	Components.P2_FixUnit
        .SuspendMoveWorkExpression( Components.P2_FixUnit.MoveWorkTask.Busy AND NOT inSafeCondition, '<#Movement is blocked due safe zone is interupted(robot in zone)#>');

    Components.P2_FixUnit
        .SuspendMoveHomeExpression(Components.P2_FixUnit.MoveHomeTask.Busy AND NOT inSafeCondition, '<#Movement is blocked due safe zone is interupted(robot in zone)#>');
END_IF;

IF _timerDisableSafety.Q THEN
	_temporarilyDisableSafety:=FALSE;
END_IF

PROPERTY Components : REFERENCE TO TcoPlbPaletizator_Components
GET
Components ref=_components;
END_GET
END_PROPERTY

(*~
	<docu>
		<summary>
			Gets the configuration of the MTS Pls feeder. 					
		</summary>			
	</docu>	
~*)
PROPERTY Config : REFERENCE TO TcoPlbPaletizator_Config_v_1_x_x
GET
Config REF= _config;
END_GET
END_PROPERTY

METHOD PUBLIC DefaultSignalisation
VAR_INPUT
END_VAR
Components.Q1_AttentionSignalisationR.Reset();
Components.Q2_AttentionSignalisationG.Reset();
Components.Q3_AttentionSignalisationB.Reset();

_blinker(inOffTime:=_config.BlinkTime,inOnTime:=_config.BlinkTime);
_timerEntryEmpty(in:= _status.EntryBufferEmpty,Pt:=_config.InfoTime);
_timerOutFull(in:=  _status.OutBufferFull ,Pt:=_config.InfoTime);
IF 
	NOT _timerEntryEmpty.Q
	AND NOT _timerOutFull.q THEN
	Components.Q2_AttentionSignalisationG.Set();
ELSIF  _blinker.IsOn THEN
	//all empty or disabled
//	IF NOT( NOT Components.I2_iBuffer1IsReadyToLoad.Signal
//		XOR NOT _config.Buffer1Disabled)
//		AND 
//		NOT(NOT Components.I4_iBuffer2IsReadyToLoad.Signal
//		XOR NOT _config.Buffer2Disabled)
//		AND
//		NOT( NOT Components.I6_iBuffer3IsReadyToLoad.Signal
//		XOR NOT _config.Buffer3Disabled)
//		AND 
//		NOT( NOT Components.I8_iBuffer4IsReadyToLoad.Signal
//		XOR NOT _config.Buffer4Disabled)
		
//		 THEN
//		Components.Q1_AttentionSignalisationR.Set();
	IF inLightCurtainOk AND 
		(
		THIS^._feedNewBlisterTask.Busy
		OR
		THIS^._throwBlisterTask.Busy
		)THEN
		Messenger.Warning('<#CAKANIE NA OBSLUHU PALETIZERA - NARUSENA SVETELNA BRANA!#>');
		Components.Q1_AttentionSignalisationR.Set();
		Components.Q2_AttentionSignalisationG.Set();
	ELSIF _timerEntryEmpty.Q
		THEN
		Components.Q1_AttentionSignalisationR.Set();
		Components.Q2_AttentionSignalisationG.Set();
	ELSIF _timerOutFull.Q
		THEN
		
		Components.Q1_AttentionSignalisationR.Set();
		Components.Q2_AttentionSignalisationG.Set();
	
//	ELSIF NOT _status.OutBufferFull
//		AND _status.EntryBufferEmpty 
//		AND NOT _status.BlisterReady THEN	
//		Components.Q1_AttentionSignalisationR.Set();
//	ELSIF  _status.OutBufferFull  THEN
//		Components.Q1_AttentionSignalisationR.Set();	
	
	END_IF;


	
END_IF;
END_METHOD

METHOD PUBLIC FeedNewBlister : TcoCore.ITcoTaskStatus

FeedNewBlister := _feedNewBlisterTask.Invoke();
END_METHOD

PROPERTY FeedNewBlisterTask : REFERENCE TO TcoFeedingSequenceTask
GET
FeedNewBlisterTask ref=_feedNewBlisterTask;
END_GET
END_PROPERTY

METHOD PUBLIC LoaadPositions : BOOL
VAR_INPUT
END_VAR
LoaadPositions:= Components.Manipulator.LoadPositionsTask.WithId(_config.PositionsSetName).Invoke().Done and Components.Manipulator.LoadPositionsTask.ReadSuccessfuly ;
END_METHOD

PROPERTY OutBufferFull : bool
GET
OutBufferFull:=_status.OutBufferFull;
END_GET
END_PROPERTY

PROPERTY ReadyToUnloadComponent : bool
GET
ReadyToUnloadComponent:=_status.ReadyToUnloadComponents;
END_GET
END_PROPERTY

(*~
	<docu>
		<summary>
			Restores this instance to the Ready state. Can be called explicitly or from within one of the restore mechanisms.	
		</summary>			
	</docu>	
~*)
METHOD  Restore : ITcoRestorable
_components.Manipulator.Restore();
_feedNewBlisterTask.Restore();
_throwBlisterTask.Restore();
_setToDefaultTask.Restore();
_messenger.UnPin();
END_METHOD

METHOD PRIVATE SequenceIncomingBlister
VAR_INPUT
	refSequenceTask : REFERENCE TO TcoFeedingSequenceTask;
	
	
END_VAR

VAR
    seq    : REFERENCE TO TcoCore.TcoSequence;


END_VAR

VAR_INST
	_timer:ton;
	_moveParam: TcoSingleAxisMoveParam;

END_VAR
seq REF= refSequenceTask.Sequence;
refSequenceTask(inoStatus := _status, inoConfig := _config);

IF NOT Components.I1_iBuffer1HasNotCriticalLevel.Signal AND NOT _config.Buffer1Disabled THEN
    Messenger.Warning('<#Buffer 1  minimalne mnozstvo!#>');
END_IF

IF NOT Components.I3_iBuffer2HasNotCriticalLevel.Signal AND NOT _config.Buffer2Disabled THEN
    Messenger.Warning('<#Buffer 2 minimalne mnozstvo!#>');
END_IF

IF NOT Components.I5_iBuffer3HasNotCriticalLevel.Signal AND NOT _config.Buffer3Disabled THEN
    Messenger.Warning('<#Buffer 3 minimalne mnozstvo!#>');
END_IF

IF NOT Components.I7_iBuffer4HasNotCriticalLevel.Signal AND NOT _config.Buffer4Disabled THEN
    Messenger.Warning('<#Buffer 4 minimalne mnozstvo!#>');
END_IF

seq.Open();
seq.Observer := refSequenceTask.Observer;

//***************************************************************************************************     
//    This step will be executed and immediately finished, as the condition in Await method is true.
IF seq.Step(0, TRUE, '<#INIT#>') THEN
    Messenger.Warning('<#BEZPECNOST ZARIADENIA NARUSENA. NIEJE MOZNE VYKONAT AKCIU#>');
    IF _status.SafeCondition THEN
        seq.CompleteStep();
    END_IF;
END_IF

//***************************************************************************************************     

//***************************************************************************************************     
IF seq.Step(20, TRUE, '<#ZASUNUTIE POZICNEJ JEDNOTKY#>') THEN

    seq.StepCompleteWhen( (*Components.P2_FixUnit.MoveToWork().Done OR*)
        Components.I11_BlisterInWorkPosition.IsFalse AND_THEN Components.P1_PositionUnit.MoveToHome().Done);

END_IF

//***************************************************************************************************     

//IF (seq.Step(inStepID := 25,
//    inEnabled := TRUE,
//    inStepDescription := 'LOAD CREATED POSITIONS')) THEN
//    //--------------------------------------------------------   
//    IF Seq.IsFreshState THEN
//        Components.Manipulator.Restore();
//    END_IF

//    IF Components.Manipulator.LoadPositionsTask.WithId(_config.PositionsSetName).Invoke().Done AND
//        Components.Manipulator.LoadPositionsTask.ReadSuccessfuly THEN
//        seq.CompleteStep();
//    END_IF

//    //--------------------------------------------------------			
//END_IF

//***************************************************************************************************     
IF seq.Step(30, TRUE, '<#KONTROLA STAVU ZASOBNIKOV') THEN

    IF Components.I2_iBuffer1IsReadyToLoad.IsTrue AND NOT _config.Buffer1Disabled THEN
        _requiredPosition := _positions.LoadFromBuffer1Pos;
        seq.StepCompleteWhen(TRUE);

    ELSIF Components.I4_iBuffer2IsReadyToLoad.Istrue AND NOT _config.Buffer2Disabled THEN
        _requiredPosition := _positions.LoadFromBuffer2Pos;
        seq.StepCompleteWhen(TRUE);

    ELSIF Components.I6_iBuffer3IsReadyToLoad.IsTrue AND NOT _config.Buffer3Disabled THEN
        _requiredPosition := _positions.LoadFromBuffer3Pos;
        seq.StepCompleteWhen(TRUE);

    ELSIF Components.I8_iBuffer4IsReadyToLoad.IsTrue AND NOT _config.Buffer4Disabled THEN
        _requiredPosition := _positions.LoadFromBuffer4Pos;
        seq.StepCompleteWhen(TRUE);
    ELSE
        IF _config.Buffer1Disabled AND _config.Buffer2Disabled AND _config.Buffer3Disabled AND _config.Buffer4Disabled THEN
            Messenger.Error('<#VSETKY ZASDOBNIKY SU VYPNUTE !!!#>');
        ELSE
            Messenger.Error('<#CHYBA ZASOBNIKY SU PRAZDNE !!!#>');

        END_IF
    END_IF
END_IF

//***************************************************************************************************     

//***************************************************************************************************     
IF seq.Step(34, TRUE, 'RESET MANIPULATORA') THEN
    IF Seq.IsFreshState OR NOT inLightCurtainOk THEN
        Components.Manipulator.Restore();
    END_IF

    IF inLightCurtainOk THEN

        IF Components.Manipulator.ResetDrive().Done AND_THEN
            Components.Manipulator.SoeReset().Done AND_THEN
            NOT Components.Manipulator.Axis.AxisStatus.Error THEN
            seq.CompleteStep();
        END_IF;
    END_IF
END_IF

//***************************************************************************************************     

//***************************************************************************************************     
IF seq.Step(35, TRUE, 'RESET MANIPULATORA') THEN
    //    IF seq.CurrentStep.Duration >= T#2S THEN
    //        seq.RequestStep(34);

    //    END_IF

    //    seq.StepCompleteWhen(Components.Manipulator.Initialize());
    Seq.CompleteStep();
END_IF

//***************************************************************************************************     

//***************************************************************************************************     
IF seq.Step(40, TRUE, 'PRESUN MANIPULATORA - NOVY BLISTER') THEN
    IF Seq.IsFreshState THEN
        Components.Manipulator.Restore();
    END_IF

    IF Components.Manipulator.Axis.AxisStatus.Error OR Components.Manipulator.Axis.AxisStatus.Disabled THEN
        seq.RequestStep(34);
    END_IF

    _moveParam.Position := _requiredPosition.Axis1.Position;
    _moveParam.Velocity := _requiredPosition.Axis1.Velocity;
    _moveParam.Acceleration := _requiredPosition.Axis1.Acceleration;
    _moveParam.Deceleration := _requiredPosition.Axis1.Deceleration;
    _moveParam.Jerk := _requiredPosition.Axis1.Jerk;

    IF Components.Manipulator.MoveAbsolute(_moveParam).Done THEN
        seq.CompleteStep();
    END_IF

END_IF

//***************************************************************************************************     

//***************************************************************************************************     
IF seq.Step(45, TRUE, 'KONTROLA BLISTRA VO FIXTURE') THEN

    Messenger.OnCondition(NOT Components.I12_BlisterPickedCorrectly.Signal).Error('<#KOLIZNY STAV SKONTROLUJTE BLISTRE!!!#>');

    seq.StepCompleteWhen(COmponents.I11_BlisterInWorkPosition.IsFalse);

END_IF

//***************************************************************************************************     

//***************************************************************************************************     
IF seq.Step(50, TRUE, 'VYSUNUTIE POZICNEJ JEDNOTKY') THEN
    IF seq.IsFreshState THEN
        _timer(IN := FALSE);
    END_IF

    _timer(IN := Components.P1_PositionUnit.MoveToWork().Done, PT := _config.StabilisationTime);
    seq.StepCompleteWhen(Components.P2_FixUnit.MoveToHome().Done AND_THEN Components.P1_PositionUnit.MoveToWork().Done AND _timer.Q);

END_IF

//***************************************************************************************************     

//***************************************************************************************************     
IF seq.Step(60, TRUE, 'UPEVNENIE BLISTRA') THEN
    IF seq.IsFreshState THEN
        _timer(IN := FALSE);
    END_IF

    _timer(IN := Components.P2_FixUnit.MoveToWork().Done, PT := _config.StabilisationTime);

    seq.StepCompleteWhen(_timer.Q);
END_IF

//***************************************************************************************************     

//***************************************************************************************************     
IF seq.Step(70, TRUE, 'ZASUNUTIE POZICNEJ JEDNOTKY A KONTROLA BLISTRA') THEN
    Messenger.OnCondition(Components.P1_PositionUnit.AtHome AND NOT Components.I11_BlisterInWorkPosition.Signal)
        .Error('NEPODARILO SA ODOBRAT BLISTER (PLNY)!');

    Messenger.OnCondition(Components.P1_PositionUnit.AtHome AND
            NOT Components.I12_BlisterPickedCorrectly.Signal).Error('<#KOLIZNY STAV SKONTROLUJTE BLISTRE!!!#>');

    IF Components.P1_PositionUnit.MoveToHome().Done AND_THEN
        Components.I11_BlisterInWorkPosition.IsTrue AND
        Components.I12_BlisterPickedCorrectly.IsTrue THEN
        seq.RequestStep(75);
    END_IF
END_IF

//***************************************************************************************************     
//***************************************************************************************************     
IF seq.Step(74, TRUE, 'RESET MANIPULATORA') THEN
    IF Seq.IsFreshState or not inLightCurtainOk THEN
        Components.Manipulator.Restore();
    END_IF

    IF inLightCurtainOk THEN
        IF Components.Manipulator.ResetDrive().Done AND_THEN
            Components.Manipulator.SoeReset().Done AND_THEN
            NOT Components.Manipulator.Axis.AxisStatus.Error THEN
            seq.CompleteStep();
        END_IF;
    END_IF;
END_IF

//***************************************************************************************************     

//***************************************************************************************************     
IF seq.Step(75, TRUE, 'RESET MANIPULATORA') THEN
    //    IF seq.CurrentStep.Duration >= T#2S THEN
    //        seq.RequestStep(34);

    //    END_IF

    //    seq.StepCompleteWhen(Components.Manipulator.Initialize());
    Seq.CompleteStep();
END_IF

//***************************************************************************************************     

//***************************************************************************************************     
IF seq.Step(80, TRUE, ' PRESUN MANIPULATORA - VYLOZENIE PRAZDNY BLISTER') THEN
    IF Seq.IsFreshState THEN
        Components.Manipulator.Restore();
    END_IF

    IF Components.Manipulator.Axis.AxisStatus.Error OR Components.Manipulator.Axis.AxisStatus.Disabled THEN
        seq.RequestStep(74);
    END_IF

    _requiredPosition := _positions.WorkPos;
    _moveParam.Position := _requiredPosition.Axis1.Position;
    _moveParam.Velocity := _requiredPosition.Axis1.Velocity;
    _moveParam.Acceleration := _requiredPosition.Axis1.Acceleration;
    _moveParam.Deceleration := _requiredPosition.Axis1.Deceleration;
    _moveParam.Jerk := _requiredPosition.Axis1.Jerk;

    IF Components.Manipulator.MoveAbsolute(_moveParam).Done THEN
        seq.CompleteStep();
    END_IF

END_IF

//***************************************************************************************************     
IF seq.Step(90, TRUE, 'VYSUNUTIE POZICNEJ JEDNOTKY') THEN

    seq.StepCompleteWhen(Components.P1_PositionUnit.MoveToWork().Done);

END_IF

//***************************************************************************************************     

IF (seq.Step(inStepID := seq.RESTORE_STEP_ID,
    inEnabled := TRUE,
    inStepDescription := 'RETURN TO THE START OF THE SEQUENCE')) THEN
    //--------------------------------------------------------	
    refSequenceTask.DoneWhen(TRUE);
    seq.CompleteSequence();
    //--------------------------------------------------------			
END_IF;

IF refSequenceTask.HandleTaskError() THEN
    //here we can decide what to do
    //	refSequenceTask.Restore();
    _feedNewBlisterTask.Restore();
END_IF

seq.Close();
END_METHOD

METHOD PRIVATE SequenceOutgoingBlister
VAR_INPUT
	refSequenceTask : REFERENCE TO TcoFeedingSequenceTask;
	
	
END_VAR

VAR
    seq    : REFERENCE TO TcoCore.TcoSequence;

END_VAR

VAR_INST
	_timer:ton;
	_timerOptional:ton;
	_moveParam: TcoSingleAxisMoveParam;

END_VAR
seq REF= refSequenceTask.Sequence;
refSequenceTask(inoStatus := _status, inoConfig := _config);

IF Components.I9_iThrowBuffer1Isfull.Signal AND NOT _config.EmptyBuffer1Disabled THEN
    Messenger.Warning('<#VYSTUPNY ZASOBNIK 1 PLNY(BUFFER) !!!#>');
END_IF

IF Components.I10_iThrowBuffer2Isfull.Signal AND NOT _config.EmptyBuffer2Disabled THEN
    Messenger.Warning('<#VYSTUPNY ZASOBNIK 2 PLNY(BUFFER) !!!#>');
END_IF

seq.Open();
seq.Observer := refSequenceTask.Observer;

//***************************************************************************************************     
//    This step will be executed and immediately finished, as the condition in Await method is true.
IF seq.Step(0, TRUE, '<#INIT#>') THEN
    Messenger.Warning('<#BEZPECNOST ZARIADENIA NARUSENA. NIEJE MOZNE VYKONAT AKCIU#>');
    IF _status.SafeCondition THEN
        seq.CompleteStep();
    END_IF;
END_IF

//***************************************************************************************************     

//***************************************************************************************************     
IF seq.Step(10, TRUE, 'ZASUNUTIE POZICNEJ JEDNOTKY') THEN

    seq.StepCompleteWhen((Components.P2_FixUnit.MoveToWork().Done OR Components.I11_BlisterInWorkPosition.IsFalse) AND_THEN
            Components.P1_PositionUnit.MoveToHome().Done);

END_IF

//***************************************************************************************************     

//IF (seq.Step(inStepID := 25,
//    inEnabled := TRUE,
//    inStepDescription := 'LOAD CREATED POSITIONS')) THEN
//    //--------------------------------------------------------   
//    IF Seq.IsFreshState THEN
//        Components.Manipulator.Restore();
//    END_IF

//    IF Components.Manipulator.LoadPositionsTask.WithId(_config.PositionsSetName).Invoke().Done AND
//        Components.Manipulator.LoadPositionsTask.ReadSuccessfuly THEN
//        seq.CompleteStep();
//    END_IF

//    //--------------------------------------------------------			
//END_IF

//***************************************************************************************************     

//***************************************************************************************************     
IF seq.Step(20, TRUE, 'KONTROLA ZASOBNIKOU PRE PRAZDNE BLISTRE') THEN

    Messenger.OnCondition(Components.I9_iThrowBuffer1Isfull.Signal AND NOT _config.EmptyBuffer1Disabled)
        .Warning('<#Zasobnik 1 na prazdne blistre plny!#>');

    Messenger.OnCondition(Components.I10_iThrowBuffer2Isfull.Signal AND NOT _config.EmptyBuffer2Disabled)
        .Warning('<#Zasobnik 2 na prazdne blistre plny!#>');

    IF Components.I9_iThrowBuffer1Isfull.IsFalse AND NOT _config.EmptyBuffer1Disabled THEN
        _requiredPosition := _positions.UnloadEmpty1Postion;
        seq.StepCompleteWhen(TRUE);

    ELSIF Components.I10_iThrowBuffer2Isfull.IsFalse AND NOT _config.EmptyBuffer2Disabled THEN
        _requiredPosition := _positions.UnloadEmpty2Postion;
        seq.StepCompleteWhen(TRUE);
    ELSE
        IF _config.EmptyBuffer1Disabled AND _config.EmptyBuffer2Disabled THEN
            Messenger.Error('<#ZASDOBNIKY PRE PRAZDNE BLISTRE SU VYPNUTE !!!#>');
        ELSE
            Messenger.Error('<#CHYBA ZASOBNIKY NA PRAZDNE BLISTRE OBSADENE !!!#>');

        END_IF
    END_IF;

END_IF

//***************************************************************************************************     

//***************************************************************************************************     
IF seq.Step(34, TRUE, 'RESET MANIPULATORA') THEN
    IF Seq.IsFreshState or not inLightCurtainOk THEN
        Components.Manipulator.Restore();
    END_IF

    IF inLightCurtainOk THEN
        IF Components.Manipulator.ResetDrive().Done AND_THEN
            Components.Manipulator.SoeReset().Done AND_THEN
            NOT Components.Manipulator.Axis.AxisStatus.Error THEN
            seq.CompleteStep();
        END_IF;
    END_IF;
END_IF

//***************************************************************************************************     

//***************************************************************************************************     
IF seq.Step(35, TRUE, 'RESET MANIPULATORA') THEN
    //    IF seq.CurrentStep.Duration >= T#2S THEN
    //        seq.RequestStep(34);

    //    END_IF

    //    seq.StepCompleteWhen(Components.Manipulator.Initialize());
    Seq.CompleteStep();
END_IF

//***************************************************************************************************     

//***************************************************************************************************     
IF seq.Step(40, TRUE, 'PRESUN MANIPULATORA - NOVY BLISTER') THEN
    IF Seq.IsFreshState THEN
        Components.Manipulator.Restore();
    END_IF

    IF Components.Manipulator.Axis.AxisStatus.Error OR Components.Manipulator.Axis.AxisStatus.Disabled THEN
        seq.RequestStep(34);
    END_IF

    _moveParam.Position := _requiredPosition.Axis1.Position;
    _moveParam.Velocity := _requiredPosition.Axis1.Velocity;
    _moveParam.Acceleration := _requiredPosition.Axis1.Acceleration;
    _moveParam.Deceleration := _requiredPosition.Axis1.Deceleration;
    _moveParam.Jerk := _requiredPosition.Axis1.Jerk;

    IF Components.Manipulator.MoveAbsolute(_moveParam).Done THEN
        seq.CompleteStep();
    END_IF

END_IF

//***************************************************************************************************    

//***************************************************************************************************     
IF seq.Step(43, TRUE, 'VYLOZENIE PRAZDNEHO BLISTRA DO ZASOBNIKA PRESUN POZICNEJ JEDNOTKY') THEN
    IF seq.IsFreshState THEN
        _timer(IN := FALSE);
    END_IF

    _timer(IN := Components.P1_PositionUnit.MoveToWork().Done, PT := _config.StabilisationTime);

    seq.StepCompleteWhen(_timer.Q);

END_IF

//***************************************************************************************************     
IF seq.Step(45, TRUE, 'VYLOZENIE PRAZDNEHO BLISTRA DO ZASOBNIKA') THEN
    IF seq.IsFreshState THEN
        _timer(IN := FALSE);
        _timerOptional(IN := FALSE);
    END_IF

    _timer(IN := Components.P2_FixUnit.MoveToHome().Done, PT := _config.StabilisationTime);
    _timerOptional(IN := Components.I11_BlisterInWorkPosition.IsFalse, PT := _config.StabilisationTime);

    seq.StepCompleteWhen(_timer.Q OR _timerOptional.Q);
END_IF

//***************************************************************************************************     
IF seq.Step(50, TRUE, 'VYLOZENIE PRAZDNEHO BLISTRA DO ZASOBNIKA') THEN

    seq.StepCompleteWhen(Components.P1_PositionUnit.MoveToHome().Done);

END_IF

//*************************************************************************************************** 

//***************************************************************************************************     
IF seq.Step(60, TRUE, 'KONTROLA VYLOZENIA BLISTRA DO  ZASOBNIKA (PRAZDNE)') THEN
    Messenger.Error('NEPODARILO SA VYLOZIT PRAZDNY BLISTER!');
    seq.StepCompleteWhen(Components.I11_BlisterInWorkPosition.IsFalse);

END_IF

//*************************************************************************************************** 

IF (seq.Step(inStepID := seq.RESTORE_STEP_ID,
    inEnabled := TRUE,
    inStepDescription := 'RETURN TO THE START OF THE SEQUENCE')) THEN
    //--------------------------------------------------------	
    refSequenceTask.DoneWhen(TRUE);
    seq.CompleteSequence();
    //--------------------------------------------------------			
END_IF;

IF refSequenceTask.HandleTaskError() THEN
    //here we can decide what to do
    //	refSequenceTask.Restore();
    _throwBlisterTask.Restore();

END_IF

seq.Close();
END_METHOD

METHOD PRIVATE SequenceSetToDefault
VAR_INPUT
	refSequenceTask : REFERENCE TO TcoFeedingSequenceTask;
	inResetOnlyManipulator:BOOL;
	
END_VAR

VAR
    seq    : REFERENCE TO TcoCore.TcoSequence;

END_VAR

VAR_INST
	_timer:ton;
	
END_VAR
seq REF= refSequenceTask.Sequence;
refSequenceTask(inoStatus:=_status,inoConfig:=_config);
seq.Open();
seq.Observer := refSequenceTask.Observer;



		



//***************************************************************************************************     
//    This step will be executed and immediately finished, as the condition in Await method is true.
IF seq.Step(0,TRUE,'<#INIT#>') THEN   
	Messenger.Warning('<#BEZPECNOST ZARIADENIA NARUSENA. NIEJE MOZNE VYKONAT AKCIU#>');     
	IF _status.SafeCondition THEN
    	seq.CompleteStep();
	END_IF;
END_IF        
//***************************************************************************************************     



//***************************************************************************************************     
IF seq.Step(10,NOT inResetOnlyManipulator,'<#VYCHODIZA POLOHA - ZASUNUTIE POZICIEJ JEDNOTKY P1 #>') THEN   

    seq.StepCompleteWhen(Components.P1_PositionUnit.MoveToHome().Done );
END_IF        
//***************************************************************************************************   


//***************************************************************************************************     
IF seq.Step(20,not inResetOnlyManipulator,'<#VYCHODIZA POLOHA - ZASUNUTIE UPEVNENIA BLISTRA  P2#>') THEN   

    seq.StepCompleteWhen(Components.P2_FixUnit.MoveToHome().Done);
END_IF        
//***************************************************************************************************   


//***************************************************************************************************     
IF (seq.Step(inStepID := 30,
    inEnabled := TRUE,
    inStepDescription := 'LOAD POSITIONS FROM DB')) THEN
    //--------------------------------------------------------   
    IF Seq.IsFreshState THEN
        Components.Manipulator.Restore();
    END_IF

    IF Components.Manipulator.LoadPositionsTask.WithId(_config.PositionsSetName).Invoke().Done AND
        Components.Manipulator.LoadPositionsTask.ReadSuccessfuly THEN
        seq.CompleteStep();
    END_IF

    //--------------------------------------------------------			
END_IF      

//***************************************************************************************************     
IF seq.Step(40, TRUE, 'RESET MANIPULATORA') THEN
    IF Seq.IsFreshState THEN
        Components.Manipulator.Restore();
    END_IF

    IF Components.Manipulator.ResetDrive().Done AND_THEN
        Components.Manipulator.SoeReset().Done AND_THEN
        NOT Components.Manipulator.Axis.AxisStatus.Error THEN
        seq.CompleteStep();
    END_IF;
END_IF

//***************************************************************************************************     




IF (seq.Step(inStepID := seq.RESTORE_STEP_ID,
    inEnabled := TRUE,
    inStepDescription := 'RETURN TO THE START OF THE SEQUENCE')) THEN
    //--------------------------------------------------------	
		refSequenceTask.DoneWhen(TRUE);
    	seq.CompleteSequence();
    //--------------------------------------------------------			
END_IF;



IF refSequenceTask.HandleTaskError() THEN
	
	//here we can decide what to do
	//	refSequenceTask.Restore();

END_IF

seq.Close();
END_METHOD

(*~
	<docu>
		<summary>
		    Custom service (manual, maintenance) logic.
			This method must be implemented in derived class.
		</summary>			
	</docu>	
~*)
METHOD PROTECTED  ServiceMode
_components.Q3_AttentionSignalisationB.Service();
_components.Q2_AttentionSignalisationG.Service();
_components.Q1_AttentionSignalisationR.Service();
_components.P2_FixUnit.Service();
_components.P1_PositionUnit .Service();
_components.Manipulator.Service();
END_METHOD

PROPERTY PUBLIC SetSequencesToStep : bool
GET
SetSequencesToStep:=_setSequencesToStep;
END_GET
SET
_setSequencesToStep:=SetSequencesToStep;
END_SET
END_PROPERTY

METHOD PUBLIC SetToDefault : TcoCore.ITcoTaskStatus

VAR
	inResetOnlyManipulator:BOOL;
END_VAR
_control.ResetOnlyManipulator:=inResetOnlyManipulator;
SetToDefault := _setToDefaultTask.Invoke();
END_METHOD

PROPERTY SetToDefaultTask : REFERENCE TO TcoFeedingSequenceTask
GET
SetToDefaultTask ref=_setToDefaultTask;
END_GET
END_PROPERTY

(*~
	<docu>
		<summary>
			Gets the status of the MTS Pls feeder. 					
		</summary>			
	</docu>	
~*)
PROPERTY Status : REFERENCE TO TcoPlbPaletizator_Status_v_1_x_x
GET
Status REF= _status;
END_GET
END_PROPERTY

METHOD PUBLIC ThrowBlister : TcoCore.ITcoTaskStatus

ThrowBlister := _throwBlisterTask.Invoke();
END_METHOD

PROPERTY ThrowBlisterTask : REFERENCE TO TcoFeedingSequenceTask
GET
ThrowBlisterTask ref=_throwBlisterTask;
END_GET
END_PROPERTY

END_FUNCTION_BLOCK

// ---- Abstractions/Components/MtsFeeding/TcoFeedingSequenceTask.TcPOU
FUNCTION_BLOCK  TcoFeedingSequenceTask EXTENDS TcoCore.TcoTask
VAR_IN_OUT
	inoStatus:TcoFeeding_Status_v_1_x_x;
	inoConfig:TcoFeeding_Config_v_1_x_x;

END_VAR
VAR
	_sequence      : TcoCore.TcoSequence(THIS^, eRestoreMode.None);
    _observerSequence       : TcoCore.TcoSequencerObserver(THIS^);
	_infoTime:TIME;
	_errorTime:	TIME;
	_errorMessage:TcoCore.TcoMessenger(THIS^);

END_VAR

IF  __ISVALIDREF(inoConfig) THEN  
_infoTime := THIS^.inoConfig.InfoTime;
_errorTime := THIS^.inoConfig.ErrorTime;
END_IF;

PROPERTY PUBLIC ErrorTime : REFERENCE TO TIME
GET
ErrorTime REF=_errorTime;
END_GET
END_PROPERTY

METHOD PUBLIC HandleTaskError :BOOL;
VAR_INPUT
END_VAR
IF THIS^.ElapsedTime > THIS^.ErrorTime AND THIS^.ErrorTime<>T#0S THEN
	THIS^.ThrowWhen(TRUE);
END_IF

HandleTaskError := THIS^.Error AND NOT THIS^._errorMessage.Pinned;
END_METHOD

PROPERTY InfoTime :REFERENCE TO TIME
GET
InfoTime REF=_infoTime;
END_GET
END_PROPERTY

PROPERTY PUBLIC Observer : REFERENCE TO TcoCore.TcoSequencerObserver
GET
Observer ref=_observerSequence;
END_GET
END_PROPERTY

METHOD PROTECTED OnError
VAR
	description: STRING;
END_VAR
description := '<#Task finished with error.#>'; 
IF  __ISVALIDREF(inoStatus) THEN   THIS^.inoStatus.ActionDescription := description; END_IF;
THIS^._errorMessage.Error('To restore acknowledge this alarm.').Pin();
END_METHOD

(*~
	<docu>
		<summary>
			Restores this instance to the Ready state. Can be called explicitly or from within one of the restore mechanisms.
			<para>
				See also <see cref="PlcDocu.TcoCore.TcoTask.AutoRestorable()"/>
			</para>
		</summary>			
	</docu>	
~*)
METHOD Restore : ITcoRestorable
SUPER^.Restore();
_sequence.ModeController.Mode :=eSequencerMode.CyclicMode;
_messenger.UnPin();
_errorMessage.UnPin();
_sequence.Restore();
END_METHOD

PROPERTY PUBLIC Sequence : REFERENCE TO TcoCore.TcoSequence
GET
Sequence ref=_sequence;
END_GET
END_PROPERTY

METHOD SetCyclicMode
VAR_INPUT
END_VAR
_sequence.ModeController.Mode :=eSequencerMode.CyclicMode;
END_METHOD

METHOD SetStepMode
VAR_INPUT
END_VAR
_sequence.ModeController.Mode :=eSequencerMode.StepMode;
END_METHOD

END_FUNCTION_BLOCK

// ---- Abstractions/Components/MtsFeeding/Blisters/Plb/TcoPlbPaletizator_Positions.TcPOU
FUNCTION_BLOCK TcoPlbPaletizator_Positions EXTENDS TcoDrivesBeckhoff.TcoSingleAxisPositionsRootContainer
VAR_INPUT
END_VAR
VAR_OUTPUT
END_VAR
VAR

	
	{attribute addProperty Name "<#Pracovna pozicia#>"}
	WorkPosition : TcoDrivesBeckhoff.TcoMultiAxisMoveParam;
	{attribute addProperty Name "<#Naberacia pozicia Buffer1#>"}
	LoadFromBuffer1Postion : TcoDrivesBeckhoff.TcoMultiAxisMoveParam;
	{attribute addProperty Name "<#Naberacia pozicia Buffer2#>"}
	LoadFromBuffer2Postion : TcoDrivesBeckhoff.TcoMultiAxisMoveParam;
	{attribute addProperty Name "<#Naberacia pozicia Buffer3#>"}
	LoadFromBuffer3Postion : TcoDrivesBeckhoff.TcoMultiAxisMoveParam;
	{attribute addProperty Name "<#Naberacia pozicia Buffer4#>"}
	LoadFromBuffer4Postion : TcoDrivesBeckhoff.TcoMultiAxisMoveParam;
	{attribute addProperty Name "<#Vykladacia pozicia pre prazdne blistre 1#>"}
	UnloadEmpty1Postion : TcoDrivesBeckhoff.TcoMultiAxisMoveParam;
	{attribute addProperty Name "<#Vykladacia pozicia pre prazdne blistre 2#>"}
	UnloadEmpty2Postion : TcoDrivesBeckhoff.TcoMultiAxisMoveParam;

END_VAR

PROPERTY PUBLIC LoadFromBuffer1Pos : reference to TcoDrivesBeckhoff.TcoMultiAxisMoveParam;
GET
LoadFromBuffer1Pos ref=LoadFromBuffer1Postion;
END_GET
END_PROPERTY

PROPERTY PUBLIC LoadFromBuffer2Pos : reference to TcoDrivesBeckhoff.TcoMultiAxisMoveParam;
GET
LoadFromBuffer2Pos ref=LoadFromBuffer2Postion;
END_GET
END_PROPERTY

PROPERTY PUBLIC LoadFromBuffer3Pos : reference to TcoDrivesBeckhoff.TcoMultiAxisMoveParam;
GET
LoadFromBuffer3Pos ref=LoadFromBuffer3Postion;
END_GET
END_PROPERTY

PROPERTY PUBLIC LoadFromBuffer4Pos : reference to TcoDrivesBeckhoff.TcoMultiAxisMoveParam;
GET
LoadFromBuffer4Pos REF=LoadFromBuffer4Postion;
END_GET
END_PROPERTY

PROPERTY PUBLIC UnloadEmpty1Pos : reference to TcoDrivesBeckhoff.TcoMultiAxisMoveParam;
GET
UnloadEmpty1Pos REF=UnloadEmpty1Postion;
END_GET
END_PROPERTY

PROPERTY PUBLIC UnloadEmpty2Pos : reference to TcoDrivesBeckhoff.TcoMultiAxisMoveParam;
GET
UnloadEmpty2Pos REF=UnloadEmpty2Postion;
END_GET
END_PROPERTY

PROPERTY PUBLIC WorkPos : reference to TcoDrivesBeckhoff.TcoMultiAxisMoveParam;
GET
WorkPos ref= WorkPosition;
END_GET
END_PROPERTY

END_FUNCTION_BLOCK

// ---- Abstractions/Components/MtsFeeding/Blisters/Plr/TcoPlrPaletizator.TcPOU
FUNCTION_BLOCK TcoPlrPaletizator EXTENDS TcoCore.TcoComponent
VAR_INPUT
    inSafeCondition : BOOL;
    inDoorOpen : BOOL;
END_VAR

VAR_OUTPUT
END_VAR
VAR
    {attribute addProperty Name "<#Config#>"}
    _config : TcoPlrPaletizator_Config_v_1_x_x;
    {attribute addProperty Name "<#Status#>"}
    {attribute clr [ReadOnly()]}
    _status : TcoPlrPaletizator_Status_v_1_x_x;
    {attribute addProperty Name "<#Control#>"}
    _control : TcoPlrPaletizator_Control_v_1_x_x;

    {attribute addProperty Name "<#Components#>"}
    _components : TcoPlrPaletizator_Components := (Parent := THIS^);

    {attribute addProperty Name "<#Poziadavka novy blister#>"}
    _feedNewBlisterTask : TcoFeedingSequenceTask(THIS^);
    {attribute addProperty Name "<#Poziadavka vylozenie blistera#>"}
    _throwBlisterTask : TcoFeedingSequenceTask(THIS^);
   {attribute addProperty Name "<#Obsluha vystupny buffer#>"}
    _handleOutgoingBufferTask : TcoFeedingSequenceTask(THIS^);
  

   {attribute addProperty Name "<#Poziadavka obsluhy vyprazdnenia vstupny buffer#>"}
    _hanldeEmptyIncommingTask : TcoFeedingSequenceTask(THIS^);
	
    {attribute addProperty Name "<#Poziadavka vychodzej polohy#>"}
    _setToDefaultTask : TcoFeedingSequenceTask(THIS^);

    {attribute addProperty Name "<#Restore#>"}
    _restoreTask : TcoCore.TcoTask(THIS^);

    timerEntryConv : TON;
    timerOutConv : TON;
    timerEmptyConv : TON;

    {attribute clr [CompilerOmits("BuilderPlainer", "BuilderOnliner","BuilderOnlinerInterface","BuilderShadowerInterface")]}
    _blinker : TcoBlinker(THIS^);
    _timerEntryEmpty : ton;
    _timerOutFull : ton;
    _timerDisableSafety : TON;
    {attribute addProperty Name "<#Temporarily disabled safety#>"}
    _temporarilyDisableSafety : BOOL;

    {attribute clr [CompilerOmits("BuilderPlainer", "BuilderOnliner","BuilderOnlinerInterface","BuilderShadowerInterface")]}
    restoreDone : BOOL;
    {attribute clr [CompilerOmits("BuilderPlainer", "BuilderOnliner","BuilderOnlinerInterface","BuilderShadowerInterface")]}
    _setSequencesToStep : BOOL := FALSE;

    _requestOutgoingEmpty : BOOL;
	_outBufferIsWaitingEmpty: BOOL;
END_VAR

_status.SafeCondition := inSafeCondition;

Context.Environment.Messaging.Resume();
_status.EntryBufferEmpty := (NOT Components.i4_PresentBlisterAtEntryStopper2.Signal AND NOT _config.PR2_StopperConveyorEntry2Disabled) AND
    NOT Components.I6_PresentBlisterAtEntryStopper3.Signal AND
    NOT Components.I8_PresentBlisterAtEntryStopper4.Signal;

_status.BlisterReady := Components.I14_PresentBlisterInLiftEnd.Signal AND Components.PR14_Lift.AtWork AND Components.PR13_CenteringBlisterInLift.AtWork;
_status.OutBufferFull := Components.I12_OutgoingBufferIsFull.Signal AND Components.I13_OutgoingConveyorIsFull.Signal;
Context.Environment.Messaging.Suspend();

IF _config.StepModeManagableFromOutside THEN
    IF _setSequencesToStep THEN
        _feedNewBlisterTask.SetStepMode();
        _throwBlisterTask.SetStepMode();
        _handleOutgoingBufferTask.SetStepMode();
        _hanldeEmptyIncommingTask.SetStepMode();
        _setToDefaultTask.SetStepMode();
    ELSE
        _feedNewBlisterTask.SetCyclicMode();
        _throwBlisterTask.SetCyclicMode();
		_handleOutgoingBufferTask.SetCyclicMode();
        _hanldeEmptyIncommingTask.SetCyclicMode();
        _setToDefaultTask.SetCyclicMode();
    END_IF
END_IF;

_feedNewBlisterTask.Enabled := NOT _throwBlisterTask.Busy;
IF (_feedNewBlisterTask.Execute()) THEN
    SequenceIncomingBlister(refSequenceTask := _feedNewBlisterTask);
END_IF;

_throwBlisterTask.Enabled := NOT _feedNewBlisterTask.Busy;
IF (_throwBlisterTask.Execute()) THEN
    SequenceOutgoingBlister(refSequenceTask := _throwBlisterTask,refOutgoingBufferTask:=_handleOutgoingBufferTask);
END_IF;

_handleOutgoingBufferTask.Enabled := TRUE;
IF (_handleOutgoingBufferTask.Execute()) THEN
    SequenceOutgoingBuffer(refSequenceTask := _handleOutgoingBufferTask);
END_IF;

_hanldeEmptyIncommingTask.Enabled := TRUE;
IF (_hanldeEmptyIncommingTask.Execute()) THEN
    SequenceEmptyIncommingBlisters(refSequenceTask := _hanldeEmptyIncommingTask);
END_IF;

_setToDefaultTask.Enabled := TRUE;
IF (_setToDefaultTask.Execute()) THEN
    SequenceResetToDefault(refSequenceTask := _setToDefaultTask);
END_IF;

//*************RESTORE********************

_restoreTask.Enabled := TRUE;

IF _restoreTask.Execute() THEN
    Restore();
    _restoreTask.DoneWhen(inCondition := TRUE);
END_IF

//****************************************


IF Components.I16_SendButton.Signal  
	AND Components.I1_PresentBlisterAtEntryStopper1.Signal
	AND NOT Components.I2_PresentBlisterAtEntryStopper1Wipa.Signal  
	AND NOT Components.I3_NotLoadedCorrectlyAtEntryStopper1.Signal THEN
	Components.PR1_StopperConveyorEntry1.MoveToHome();
	Components.Q4_EntryConvRun.Set(); 
END_IF

IF Components.Q4_EntryConvRun.Signal 
	AND NOT Components.I16_SendButton.Signal 
	AND NOT Components.I1_PresentBlisterAtEntryStopper1.Signal THEN
		Components.PR1_StopperConveyorEntry1.MoveToWork();
END_IF

IF NOT Components.I17_EmptyButton.Signal
	and	_requestOutgoingEmpty
	AND Components.Q6_OutgoingConvRun.Signal 
	AND Components.PR5_StopperConveyorOutgoing1.AtHome
	AND NOT Components.I10_PresentBlisterAtOutgoingStopper1.Signal
	AND  NOT Components.I11_PresentBlisterAtOutgoingStopper1Wipa.Signal THEN
	Components.PR5_StopperConveyorOutgoing1.MoveToWork();
	_requestOutgoingEmpty:=false;
END_IF

IF Components.I17_EmptyButton.Signal THEN
	Components.PR5_StopperConveyorOutgoing1.MoveToHome();
	_requestOutgoingEmpty:=true;
	Components.Q6_OutgoingConvRun.Set(); 
END_IF



timerEntryConv(In:= Components.Q4_EntryConvRun.Signal OR Components.Q5_EntryConvRunReverse.Signal  ,Pt:=_config.ConveyorEntryRunTime);
timerOutConv(In:= Components.Q6_OutgoingConvRun.Signal,Pt:=_config.ConveyorOutRunTime);


Messenger.OnCondition(_config.ConveyorEntryRunTime=T#0S).Warning('<#No timeout defined for Entry conveyor running.#>');
Messenger.OnCondition(_config.ConveyorEntryRunTime=T#0S).Warning('<#No timeout defined for Our conveyor running.#>');



IF timerEntryConv.Q THEN
	Components.Q4_EntryConvRun.Reset(); 
	Components.Q5_EntryConvRunReverse.Reset(); 
	Components.Q8_LiftConvRun.Reset();
	Components.Q9_LiftConvRunReverse.Reset();

END_IF
IF timerOutConv.Q THEN
	Components.Q6_OutgoingConvRun.Reset(); 
	Components.Q7_OutgoingConvRunReverse.Reset(); 
END_IF







//********************SAFETY******************
_timerDisableSafety(IN := _temporarilyDisableSafety, PT := _config.TimeToDisableSafety);

THIS^.Messenger.OnCondition(inCondition := _temporarilyDisableSafety).Warning('SAFTY TEMPORARILY DISABLED!');

IF NOT _temporarilyDisableSafety THEN
	
	


    Components.PR14_Lift
        .SuspendMoveWorkExpression(Components.PR14_Lift.MoveWorkTask.Busy AND NOT inSafeCondition, '<#Movement is blocked due safe zone is interupted(robot in zone)#>');

    Components.PR14_Lift
        .SuspendMoveHomeExpression(Components.PR14_Lift.MoveHomeTask.Busy AND NOT inSafeCondition,'<#Movement is blocked due safe zone is interupted(robot in zone)#>');
	
    Components.PR13_CenteringBlisterInLift
        .SuspendMoveWorkExpression(Components.PR13_CenteringBlisterInLift.MoveWorkTask.Busy AND NOT inSafeCondition, '<#Movement is blocked due safe zone is interupted(robot in zone)#>');

    Components.PR13_CenteringBlisterInLift
        .SuspendMoveHomeExpression(Components.PR13_CenteringBlisterInLift.MoveHomeTask.Busy AND NOT inSafeCondition,'<#Movement is blocked due safe zone is interupted(robot in zone)#>');



END_IF;

IF _timerDisableSafety.Q THEN
    _temporarilyDisableSafety := FALSE;
END_IF

PROPERTY Components : REFERENCE TO TcoPlrPaletizator_Components
GET
Components ref=_components;
END_GET
END_PROPERTY

(*~
	<docu>
		<summary>
			Gets the configuration of the MTS Pls feeder. 					
		</summary>			
	</docu>	
~*)
PROPERTY Config : REFERENCE TO TcoPlrPaletizator_Config_v_1_x_x
GET
Config REF= _config;
END_GET
END_PROPERTY

METHOD PUBLIC DefaultSignalisation
VAR_INPUT
END_VAR
Components.Q1_AttentionSignalisationR.Reset();
Components.Q2_AttentionSignalisationG.Reset();
Components.Q3_AttentionSignalisationB.Reset();

_blinker(inOffTime:=_config.BlinkTime,inOnTime:=_config.BlinkTime);
_timerEntryEmpty(in:= _status.EntryBufferEmpty,Pt:=_config.InfoTime);
_timerOutFull(in:=  _status.OutBufferFull ,Pt:=_config.InfoTime);
IF NOT inDoorOpen  
	AND NOT _timerEntryEmpty.Q
	AND NOT _timerOutFull.q THEN
	Components.Q2_AttentionSignalisationG.Set();
ELSIF  _blinker.IsOn THEN
	IF inDoorOpen AND 
		(
		THIS^._feedNewBlisterTask.Busy
		OR
		THIS^._throwBlisterTask.Busy
		OR
		THIS^._hanldeEmptyIncommingTask.Busy )THEN
		Messenger.Warning('<#CAKANIE NA OBSLUHU PALETIZERA - ZAVRITE DVERE!#>');
		Components.Q1_AttentionSignalisationR.Set();
		Components.Q2_AttentionSignalisationG.Set();
	ELSIF _timerEntryEmpty.Q
		THEN
		Components.Q1_AttentionSignalisationR.Set();
		Components.Q2_AttentionSignalisationG.Set();
	ELSIF _timerOutFull.Q
		THEN
		
		Components.Q1_AttentionSignalisationR.Set();
		Components.Q2_AttentionSignalisationG.Set();

//	ELSIF NOT _status.OutBufferFull
//		AND _status.EntryBufferEmpty 
//		AND NOT _status.BlisterReady THEN	
//		Components.Q1_AttentionSignalisationR.Set();
//	ELSIF  _status.OutBufferFull  THEN
//		Components.Q1_AttentionSignalisationR.Set();	
	
	END_IF;


	
END_IF;
END_METHOD

METHOD PUBLIC EmptyIncommingBuffer : TcoCore.ITcoTaskStatus
EmptyIncommingBuffer := _hanldeEmptyIncommingTask.Invoke();
END_METHOD

METHOD PUBLIC FeedNewBlister : TcoCore.ITcoTaskStatus
FeedNewBlister := _feedNewBlisterTask.Invoke();
END_METHOD

PROPERTY FeedNewBlisterTask : REFERENCE TO TcoFeedingSequenceTask
GET
FeedNewBlisterTask ref=_feedNewBlisterTask;
END_GET
END_PROPERTY

PROPERTY HandleEmptyIncomingTask : REFERENCE TO TcoFeedingSequenceTask
GET
HandleEmptyIncomingTask ref=_hanldeEmptyIncommingTask;
END_GET
END_PROPERTY

PROPERTY HandleOutBufferTask : REFERENCE TO TcoFeedingSequenceTask
GET
HandleOutBufferTask ref=_hanldeEmptyIncommingTask;
END_GET
END_PROPERTY

PROPERTY OutBufferFull : bool
GET
OutBufferFull:=_status.OutBufferFull;
END_GET
END_PROPERTY

PROPERTY ReadyToUnloadComponent : bool
GET
ReadyToUnloadComponent:=_status.BlisterReady;
END_GET
END_PROPERTY

(*~
	<docu>
		<summary>
			Restores this instance to the Ready state. Can be called explicitly or from within one of the restore mechanisms.	
		</summary>			
	</docu>	
~*)
METHOD  Restore : ITcoRestorable

_hanldeEmptyIncommingTask.Restore();
_feedNewBlisterTask.Restore();
_throwBlisterTask.Restore();
_handleOutgoingBufferTask.Restore();

_setToDefaultTask.Restore();
_outBufferIsWaitingEmpty:=FALSE;

_messenger.UnPin();
END_METHOD

METHOD PRIVATE SequenceEmptyIncommingBlisters
VAR_INPUT
	refSequenceTask : REFERENCE TO TcoFeedingSequenceTask;
	
	
END_VAR

VAR
    seq    : REFERENCE TO TcoCore.TcoSequence;

END_VAR

VAR_INST
	_timer:ton;
	
END_VAR
seq REF= refSequenceTask.Sequence;
refSequenceTask(inoStatus := _status, inoConfig := _config);

seq.Open();
seq.Observer := refSequenceTask.Observer;

//***************************************************************************************************     
//    This step will be executed and immediately finished, as the condition in Await method is true.
IF seq.Step(0, TRUE, '<#INIT#>') THEN
    Messenger.Warning('<#BEZPECNOST ZARIADENIA NARUSENA. NIEJE MOZNE VYKONAT AKCIU#>');
    IF _status.SafeCondition THEN
        seq.CompleteStep();
    END_IF;
END_IF

//***************************************************************************************************     

//***************************************************************************************************     
IF seq.Step(10, true, 'ZASUNUTIE ZARAZIEK') THEN
    If Components.PR1_StopperConveyorEntry1.MoveToHome().Done AND
        (Components.PR2_StopperConveyorEntry2.MoveToHome().Done OR _config.PR2_StopperConveyorEntry2Disabled) AND
        Components.PR3_StopperConveyorEntry3.MoveToHome().Done AND
        Components.PR4_StopperConveyorEntry4.MoveToHome().Done AND
        Components.PR5_StopperConveyorOutgoing1.MoveToHome().Done then
        seq.CompleteStep();
    End_if;

END_IF

//***************************************************************************************************     

//***************************************************************************************************     
IF seq.Step(20, true, 'UVOLNENIE KUSOV V SEPARATORE') THEN
    IF Components.PR6_HorizontalSepareEntyBlisters.MoveToHome().Done AND_THEN
        Components.PR8_VerticalSepareEntryBlister1.MoveToWork().Done AND_THEN
        Components.PR9_VerticalSepareEntryBlister2.MoveToWork().Done AND_THEN
        (Components.PR12_HorizontalHoldEntryBlister.MoveToHome().Done OR _config.PR12_HorizontalHoldEntryBlisterDisabled) then
        seq.CompleteStep();
    END_IF;
END_IF

//***************************************************************************************************     

//***************************************************************************************************     
IF seq.Step(30, true, 'UVOLNENIE BLISTRU NA VYTAHU') THEN
    seq.StepCompleteWhen(Components.PR14_Lift.MoveToWork().Done AND_THEN Components.PR13_CenteringBlisterInLift.MoveToHome().Done);
END_IF

//***************************************************************************************************     

//***************************************************************************************************     
IF seq.Step(100, TRUE, 'ZAPNUTIE DOPRAVNIKOV') THEN

    seq.StepCompleteWhen(Components.Q4_EntryConvRun.Reset() AND
            Components.Q5_EntryConvRunReverse.Set() AND
            Components.Q8_LiftConvRun.Reset() AND
            Components.Q9_LiftConvRunReverse.Set());
END_IF

//***************************************************************************************************     

//***************************************************************************************************     
IF seq.Step(120, TRUE, 'KONTROLA ODOBRATIA BLISTROV NA HORNOM DOPRAVNIKU') THEN
    IF seq.IsFreshState THEN
        _timer(IN := FALSE);
    END_IF

    Components.Q4_EntryConvRun.Reset();
    Components.Q5_EntryConvRunReverse.Set();
    Components.Q8_LiftConvRun.Reset();
    Components.Q9_LiftConvRunReverse.Set();
    IF Components.I1_PresentBlisterAtEntryStopper1.IsFalse and
        Components.I2_PresentBlisterAtEntryStopper1Wipa.IsFalse and
        ((Components.i4_PresentBlisterAtEntryStopper2.IsFalse and Components.i5_PresentBlisterAtEntryStopper2Wipa.IsFalse) or
        _config.PR2_StopperConveyorEntry2Disabled) and
        Components.I6_PresentBlisterAtEntryStopper3.IsFalse and
        Components.I7_PresentBlisterAtEntryStopper3Wipa.IsFalse and
        Components.I8_PresentBlisterAtEntryStopper4.IsFalse and
        Components.I9_PresentBlisterAtEntryStopper4Wipa.IsFalse and
        Components.I14_PresentBlisterInLiftEnd.IsFalse AND
        Components.I15_PresentBlisterInLiftEntry.IsFalse THEN
        _timer(in := TRUE, Pt := T#5S);
        IF _timer.Q THEN
            seq.CompleteStep();
        END_IF;
    END_IF;
END_IF

//***************************************************************************************************     

//***************************************************************************************************     
IF seq.Step(130, TRUE, 'VYSUNUTIE ZARAZIEK') THEN
    IF seq.IsFreshState THEN
        _timer(IN := FALSE);
    END_IF

    IF Components.PR1_StopperConveyorEntry1.MoveToWork().Done AND
        (Components.PR2_StopperConveyorEntry2.MoveToWork().Done OR _config.PR2_StopperConveyorEntry2Disabled) AND
        Components.PR3_StopperConveyorEntry3.MoveToWork().Done AND
        Components.PR4_StopperConveyorEntry4.MoveToWork().Done AND
        Components.PR5_StopperConveyorOutgoing1.MoveToWork().Done THEN
        _timer(in := TRUE, Pt := T#1S);
        IF _timer.Q THEN
            seq.CompleteStep();
        END_IF;
    end_if;
END_IF

//***************************************************************************************************     

//***************************************************************************************************     
IF seq.Step(300, TRUE, 'RESET SEPARATORA') THEN

    seq.StepCompleteWhen(Components.PR6_HorizontalSepareEntyBlisters.MoveToHome().Done AND_THEN
            Components.PR8_VerticalSepareEntryBlister1.MoveToWork().Done AND_THEN
            Components.PR9_VerticalSepareEntryBlister2.MoveToWork().Done AND_THEN
            (Components.PR12_HorizontalHoldEntryBlister.MoveToHome().Done OR _config.PR12_HorizontalHoldEntryBlisterDisabled));

END_IF

//***************************************************************************************************     
//***************************************************************************************************     
IF seq.Step(310, true, 'RESET  VYTAHU') THEN
    seq.StepCompleteWhen(Components.PR14_Lift.MoveToWork().Done AND_THEN Components.PR13_CenteringBlisterInLift.MoveToWork().Done);
END_IF

//***************************************************************************************************   
//***************************************************************************************************     
IF seq.Step(320, true, 'KONTROLA POZICIE KLUCIKA') THEN
    Messenger.Warning('<#KLUCIK NIE JE VO VYCHODZEJ POZICII!#>');

    seq.StepCompleteWhen(Components.I18_EmptyKey.IsFalse);
END_IF

//***************************************************************************************************   

IF (seq.Step(inStepID := seq.RESTORE_STEP_ID,
    inEnabled := TRUE,
    inStepDescription := 'RETURN TO THE START OF THE SEQUENCE')) THEN
    //--------------------------------------------------------	
    refSequenceTask.DoneWhen(TRUE);
    seq.CompleteSequence();
    //--------------------------------------------------------			
END_IF;

IF refSequenceTask.HandleTaskError() THEN
    //here we can decide what to do
    //refSequenceTask.Restore();
    _hanldeEmptyIncommingTask.Restore();
END_IF

seq.Close();
END_METHOD

METHOD PRIVATE SequenceIncomingBlister
VAR_INPUT
    refSequenceTask : REFERENCE TO TcoFeedingSequenceTask;
  

END_VAR

VAR
    seq : REFERENCE TO TcoCore.TcoSequence;


    entrySequencer : INT;
END_VAR

VAR_INST
    _timer : ton;
    _timerOptional : ton;
END_VAR
seq REF= refSequenceTask.Sequence;
refSequenceTask(inoStatus := _status, inoConfig := _config);


seq.Open();
seq.Observer := refSequenceTask.Observer;

//***************************************************************************************************     
IF seq.Step(0, TRUE, '<#INIT#>') THEN
        seq.CompleteStep();
END_IF

//***************************************************************************************************     

//***************************************************************************************************     
IF seq.Step(5, TRUE, 'KONTROLA KLUCIK') THEN
    
    IF Components.I18_EmptyKey.Signal THEN
        Messenger.Warning('<#KLUCIK NIE JE VO VYCHODZEJ POZICII!#>');
    End_if;

    seq.StepCompleteWhen(Components.I18_EmptyKey.IsFalse);
END_IF

//***************************************************************************************************     


//***************************************************************************************************     
IF seq.Step(10, NOT _config.PR2_StopperConveyorEntry2Disabled, 'KONTROLA VSTUPNYCH BLISTROV NA ZARAZKE PR2') THEN
    Messenger.Warning('<#CAKAM NA NALOZENIE BLISTROV#>');
    IF THIS^.Components.i4_PresentBlisterAtEntryStopper2.IsTrue
		AND Components.I6_PresentBlisterAtEntryStopper3.IsFalse
		AND NOT _config.PR2_StopperConveyorEntry2Disabled	 THEN
        seq.CompleteStep();
    ELSIF THIS^.Components.I6_PresentBlisterAtEntryStopper3.IsTrue
		OR THIS^.Components.I8_PresentBlisterAtEntryStopper4.IsTrue
        THEN
        seq.RequestStep(100);
    END_IF;
END_IF

//***************************************************************************************************   
////***************************************************************************************************     
IF seq.Step(20, NOT _config.PR2_StopperConveyorEntry2Disabled, 'KONTROLA VSTUPNYCH BLISTROV NA ZARAZKE PR2') THEN
    IF seq.IsFreshState THEN
        _timer(IN := FALSE);
    END_IF

    IF Components.PR2_StopperConveyorEntry2.MoveToHome().Done AND
        Components.PR3_StopperConveyorEntry3.MoveToWork().Done AND_THEN
        Components.Q4_EntryConvRun.Set() AND_THEN
        THIS^.Components.I6_PresentBlisterAtEntryStopper3.IsTrue THEN
        _timer(IN := THIS^.Components.I6_PresentBlisterAtEntryStopper3.Signal, PT := _config.StabilisationTime);
        IF _timer.Q THEN
            seq.CompleteStep();
        END_IF;
    END_IF;
END_IF

////*************************************************************************************************** 


////***************************************************************************************************     
IF seq.Step(30, NOT _config.PR2_StopperConveyorEntry2Disabled, 'VYSUNUTIE ZARAZKY PR2') THEN
    IF THIS^.Components.PR2_StopperConveyorEntry2.MoveToWork().Done THEN
        seq.CompleteStep();
    END_IF
END_IF

//***************************************************************************************************   


//***************************************************************************************************     
IF seq.Step(100, TRUE, 'KONTROLA VSTUPNYCH BLISTROV NA ZARAZKE PR3') THEN
    Messenger.Warning('<#CAKAM NA NALOZENIE BLISTROV#>');
    Components.Q4_EntryConvRun.Set();

   IF THIS^.Components.I6_PresentBlisterAtEntryStopper3.IsTrue AND
        Components.I7_PresentBlisterAtEntryStopper3Wipa.IsFalse  AND
		Components.I8_PresentBlisterAtEntryStopper4.isFalse THEN
        seq.CompleteStep();
    ELSIF Components.I8_PresentBlisterAtEntryStopper4.IsTrue THEN //jump only if in separing position are blisters
        seq.RequestStep(300);
	ELSE
		seq.RequestStep(10);

    END_IF;
END_IF

//***************************************************************************************************     







//***************************************************************************************************     
IF seq.Step(120, TRUE, 'KONTROLA VSTUPNYCH BLISTROV NA ZARAZKE PR3') THEN
    IF seq.IsFreshState THEN
        _timer(IN := FALSE);
    END_IF

    IF Components.PR3_StopperConveyorEntry3.MoveToHome().Done AND_THEN
        Components.Q4_EntryConvRun.Set() AND_THEN
        THIS^.Components.I6_PresentBlisterAtEntryStopper3.IsFalse THEN
        _timer(IN := NOT THIS^.Components.I6_PresentBlisterAtEntryStopper3.Signal, PT := _config.StabilisationTime);
        IF _timer.Q THEN
            seq.CompleteStep();
        END_IF;
    END_IF;
END_IF

//***************************************************************************************************     

//***************************************************************************************************     
IF seq.Step(130, TRUE, 'VYSUNUTIE ZARAZKY PR3') THEN
    seq.StepCompleteWhen(THIS^.Components.PR3_StopperConveyorEntry3.MoveToWork().Done);
END_IF




/////////////////////SEPARATOR - >  VYTAH ///////////////////////////////////////
						
 
//***************************************************************************************************     
IF seq.Step(300, TRUE, 'CAKANIE NA PALETY V POZICII SEPAROVANIA PR4') THEN
    IF seq.IsFreshState THEN
        _timer(IN := FALSE);
        _timerOptional(IN := FALSE);

    END_IF

    IF THIS^.Components.I8_PresentBlisterAtEntryStopper4.Signal THEN
        _timer(IN := THIS^.Components.I8_PresentBlisterAtEntryStopper4.Signal, PT := _config.StabilisationTime);
        IF _timer.Q THEN
            seq.CompleteStep();
        END_IF;
    ELSE

        _timer(IN := TRUE, PT := T#5S);

        IF _timerOptional.Q THEN
            //            IF NOT _config.PR2_StopperConveyorEntry2Disabled THEN
            //                seq.RequestStep(10);
            //            ELSE
            seq.RequestStep(100);
            // END_IF
        END_IF;
    END_IF;

END_IF

//***************************************************************************************************     
//***************************************************************************************************     
IF seq.Step(310, NOT _config.PR12_HorizontalHoldEntryBlisterDisabled, 'PRIDLZIAVANIE BLISTRA VYSUNUT PR12') THEN
    seq.StepCompleteWhen(Components.PR12_HorizontalHoldEntryBlister.MoveToWork().Done);
END_IF

//***************************************************************************************************   

//***************************************************************************************************     
IF seq.Step(320, TRUE, 'SEPAROVANIE BLISTRA UCHOPENIE  PR9 VYSUNUT PR8 ZASUNUT A NASLEDNE PR6 VYSUNUT') THEN
    seq.StepCompleteWhen(Components.PR9_VerticalSepareEntryBlister2.MoveToWork().Done AND
            Components.PR8_VerticalSepareEntryBlister1.MoveToHome().Done AND_THEN
            Components.PR6_HorizontalSepareEntyBlisters.MoveToWork().Done);
END_IF

//***************************************************************************************************     

//***************************************************************************************************     
IF seq.Step(330, TRUE, 'SEPAROVANIE BLISTRA NADVIHNUTIE PR8 ZASUNUT PR9 ZASUNUT A NASLEDNE PR12 ZASUNUT') THEN
    seq.StepCompleteWhen(Components.PR8_VerticalSepareEntryBlister1.MoveToHome().Done AND
            Components.PR9_VerticalSepareEntryBlister2.MoveToHome().Done and_then
            Components.PR12_HorizontalHoldEntryBlister.MoveToHome().Done);
END_IF

//***************************************************************************************************     



//***************************************************************************************************     
IF seq.Step(340, TRUE, 'KONTROLA POZICIE VYAHU') THEN
    Messenger.Warning('<#VYTAH NIEJE V POZICII ALEBO JE OBSADENY#>');
    seq.StepCompleteWhen(
			Components.PR14_Lift.AtWork AND
            Components.I14_PresentBlisterInLiftEnd.IsFalse AND
            Components.I15_PresentBlisterInLiftEntry.IsFalse);
END_IF

//***************************************************************************************************    

//***************************************************************************************************     
IF seq.Step(350, TRUE, 'ZASUNUTIE CENTROVANIA (PR13)') THEN
    seq.StepCompleteWhen(Components.PR13_CenteringBlisterInLift.MoveToHome().Done);
END_IF

//***************************************************************************************************     

//***************************************************************************************************     
IF seq.Step(360, TRUE, 'ZASUNUTIE ZARAZKY PR4 A ZAPNUTIE DOPRAVNIKA') THEN

    seq.StepCompleteWhen(Components.PR4_StopperConveyorEntry4.MoveToHome().Done AND_THEN
            Components.Q4_EntryConvRun.Set() AND
            Components.Q8_LiftConvRun.Set() AND_THEN
            Components.I8_PresentBlisterAtEntryStopper4.IsFalse);

END_IF

//***************************************************************************************************    
IF seq.Step(362, TRUE, 'VYSUNUTIE ZARAZKY PR4') THEN
    IF seq.IsFreshState THEN
        _timer(IN := FALSE);
    END_IF

    Components.Q4_EntryConvRun.Set();
    Components.Q8_LiftConvRun.Set();

    IF Components.I9_PresentBlisterAtEntryStopper4Wipa.IsFalse AND_THEN
        Components.PR4_StopperConveyorEntry4.MoveToWork().Done AND_THEN
        (Components.PR8_VerticalSepareEntryBlister1.MoveToWork().Done AND Components.PR9_VerticalSepareEntryBlister2.MoveToWork().Done) AND_THEN
        Components.PR6_HorizontalSepareEntyBlisters.MoveToHome().Done THEN
        seq.CompleteStep();

    END_IF;
END_IF

////***************************************************************************************************  


////***************************************************************************************************  

IF seq.Step(370, TRUE, 'VYSUNUTIE ZARAZKY PR4  CAKANIE NA BLISTER V POZICII VYTAHU') THEN
    IF seq.IsFreshState THEN
        _timer(IN := FALSE);
    END_IF

    Components.Q4_EntryConvRun.Set();
    Components.Q8_LiftConvRun.Set();

    IF Components.I9_PresentBlisterAtEntryStopper4Wipa.IsFalse AND_THEN
        Components.PR4_StopperConveyorEntry4.MoveToWork().Done THEN
        _timer(IN := THIS^.Components.I14_PresentBlisterInLiftEnd.IsTrue, PT := _config.StabilisationTime);

        IF _timer.Q THEN
            seq.CompleteStep();
        END_IF
    END_IF;
END_IF

//***************************************************************************************************     

//***************************************************************************************************     
IF seq.Step(380, TRUE, 'VYSUNUTIE CENTROVANIA NA VYTAHU PR13 A VYPNUTIE MOTORA A ZASUNUTIE PR8') THEN

    seq.StepCompleteWhen(Components.PR8_VerticalSepareEntryBlister1.MoveToHome().Done AND
            Components.PR13_CenteringBlisterInLift.MoveToWork().Done AND_THEN
            Components.Q8_LiftConvRun.Reset());
END_IF

//***************************************************************************************************     

IF (seq.Step(inStepID := seq.RESTORE_STEP_ID,
    inEnabled := TRUE,
    inStepDescription := 'RETURN TO THE START OF THE SEQUENCE')) THEN
    //--------------------------------------------------------	
    refSequenceTask.DoneWhen(TRUE);
    seq.CompleteSequence();
    //--------------------------------------------------------			
END_IF;

IF refSequenceTask.HandleTaskError() THEN
    //here we can decide what to do
    //	refSequenceTask.Restore();
    _feedNewBlisterTask.Restore();
END_IF

seq.Close();
END_METHOD

METHOD PRIVATE SequenceOutgoingBlister
VAR_INPUT
	refSequenceTask : REFERENCE TO TcoFeedingSequenceTask;
	refOutgoingBufferTask : REFERENCE TO TcoFeedingSequenceTask;
	
	
END_VAR

VAR
    seq    : REFERENCE TO TcoCore.TcoSequence;

END_VAR

VAR_INST
	_timer:ton;
	_outgoingBufferTask : REFERENCE TO TcoFeedingSequenceTask;
END_VAR
seq REF= refSequenceTask.Sequence;
refSequenceTask(inoStatus := _status, inoConfig := _config);
_outgoingBufferTask REF= refOutgoingBufferTask;

seq.Open();
seq.Observer := refSequenceTask.Observer;

//***************************************************************************************************    
IF seq.Step(0, TRUE, '<#INIT#>') THEN

    Messenger.Warning('<#BEZPECNOST ZARIADENIA NARUSENA. NIEJE MOZNE VYKONAT AKCIU#>');

    IF _status.SafeCondition THEN
        seq.CompleteStep();

    END_IF;
END_IF

//***************************************************************************************************     

//***************************************************************************************************     
IF seq.Step(10, TRUE, 'ZASUNUTIE CENTROVANIA NA VYTAHU PR13') THEN
    IF Components.I14_PresentBlisterInLiftEnd.IsFalse AND Components.I15_PresentBlisterInLiftEntry.IsFalse THEN
        seq.RequestStep(100);
    ELSE

        seq.StepCompleteWhen(Components.Q8_LiftConvRun.Reset() AND
                Components.Q9_LiftConvRunReverse.Reset() AND_THEN
                THIS^.Components.PR13_CenteringBlisterInLift.MoveToHome().Done);
    END_IF;
END_IF

//***************************************************************************************************   

//***************************************************************************************************     
IF seq.Step(14, TRUE, '<#CAKANIE NA DOKONCENIE VYSTUPNEHO BUFFERA#>') THEN

    IF NOT _outgoingBufferTask.Busy THEN
        seq.CompleteStep();
    END_IF;
END_IF

//***************************************************************************************************   

//***************************************************************************************************     
IF seq.Step(15, TRUE, '<#START OBSLUHY VYSTUPNEHO BUFFERA#>') THEN
    IF seq.IsFreshState THEN
        _outgoingBufferTask.Restore();
    END_IF

    _outgoingBufferTask.Invoke();

    IF _outgoingBufferTask.Busy THEN
        seq.CompleteStep();

    END_IF;
END_IF

//***************************************************************************************************     

//***************************************************************************************************     
IF seq.Step(20, TRUE, 'VYTAH DOLNA POLOHA PR15 A VYSUNUTIE PR5 ') THEN

    seq.StepCompleteWhen(Components.PR14_Lift.MoveToHome().Done);
END_IF

//***************************************************************************************************   

//***************************************************************************************************     
IF seq.Step(40, TRUE, 'KONTROLA PRIPRAVENOSTI VYSTUPNEHO BUFFERA') THEN
    IF _outBufferIsWaitingEmpty AND _outgoingBufferTask.Busy THEN
        seq.CompleteStep();
    END_IF
END_IF

//***************************************************************************************************   

//***************************************************************************************************     
IF seq.Step(50, TRUE, 'ODOSLANIE BLISTRU Z VYTAHU') THEN
    IF seq.IsFreshState THEN
        _timer(IN := FALSE);
    END_IF

    IF Components.Q9_LiftConvRunReverse.Set() THEN
        _timer(in := Components.I14_PresentBlisterInLiftEnd.IsFalse AND Components.I15_PresentBlisterInLiftEntry.IsFalse,
            Pt := _config.StabilisationTime);

        IF _timer.Q  and not _outBufferIsWaitingEmpty THEN
            seq.CompleteStep();
        END_IF;
    END_IF;

END_IF

//***************************************************************************************************   

//***************************************************************************************************     
IF seq.Step(100, TRUE, 'CAKANIE NA VYTAH V HORENEJ POZICII PR14') THEN
    IF seq.IsFreshState THEN
        _timer(IN := FALSE);
    END_IF

    IF Components.PR14_Lift.MoveToWork().Busy AND Components.Q9_LiftConvRunReverse.Reset() THEN
        seq.CompleteStep();
    END_IF;
END_IF

//***************************************************************************************************   

//***************************************************************************************************   

IF (seq.Step(inStepID := seq.RESTORE_STEP_ID,
    inEnabled := TRUE,
    inStepDescription := 'RETURN TO THE START OF THE SEQUENCE')) THEN
    //--------------------------------------------------------	
    refSequenceTask.DoneWhen(TRUE);
    seq.CompleteSequence();
    //--------------------------------------------------------			
END_IF;

IF refSequenceTask.HandleTaskError() THEN
    //here we can decide what to do
    //	refSequenceTask.Restore();
    _throwBlisterTask.Restore();

END_IF

seq.Close();
END_METHOD

METHOD PRIVATE SequenceOutgoingBuffer
VAR_INPUT
	refSequenceTask : REFERENCE TO TcoFeedingSequenceTask;
	
	
END_VAR

VAR
    seq    : REFERENCE TO TcoCore.TcoSequence;

END_VAR

VAR_INST
	_timer:ton;
	
END_VAR
seq REF= refSequenceTask.Sequence;
refSequenceTask(inoStatus := _status, inoConfig := _config);

seq.Open();
seq.Observer := refSequenceTask.Observer;

//***************************************************************************************************     
//    This step will be executed and immediately finished, as the condition in Await method is true.
IF seq.Step(0, TRUE, '<#INIT#>') THEN
    seq.CompleteStep();
END_IF

//***************************************************************************************************     

//***************************************************************************************************     
IF seq.Step(10, TRUE, 'UCHOPENIE VYSTUPNYCH BLISTROV PR10 PR11 VYSUNUT') THEN

    seq.StepCompleteWhen(Components.PR10_VerticalSepareOutgoingBlister1.MoveToWork().Done AND
            Components.PR11_VerticalSepareOutgoingBlister2.MoveToWork().Done);
END_IF

//***************************************************************************************************   

//***************************************************************************************************     
IF seq.Step(20, TRUE, 'UCHOPENIE VYSTUPNYCH BLISTROV  PR7 VYSUNUT') THEN

    seq.StepCompleteWhen(Components.PR7_HorizontalSepareOutgoingBlisters.MoveToWork().Done);
END_IF

//***************************************************************************************************   

//***************************************************************************************************     
IF seq.Step(25, NOT _config.UseAutoHidePr5Dispabled, 'ZASUNUTIE ZARAZKY PR5') THEN

    seq.StepCompleteWhen(Components.PR5_StopperConveyorOutgoing1.MoveToHome().Done);
END_IF

//***************************************************************************************************   

//***************************************************************************************************     
IF seq.Step(30, TRUE, 'NADVIHNUTIE VYSTUPNYCH BLISTROV PR10 PR11 ZASUNUT') THEN

    seq.StepCompleteWhen(Components.PR10_VerticalSepareOutgoingBlister1.MoveToHome().Done AND
            Components.PR11_VerticalSepareOutgoingBlister2.MoveToHome().Done);
END_IF

//***************************************************************************************************   

//***************************************************************************************************     
IF seq.Step(40, TRUE, 'VYSUNUTIE ZARAZKY PR5') THEN

    seq.StepCompleteWhen(Components.PR5_StopperConveyorOutgoing1.MoveToWork().Done AND Components.I10_PresentBlisterAtOutgoingStopper1.IsFalse);
END_IF

//***************************************************************************************************   

_outBufferIsWaitingEmpty:=FALSE;

//***************************************************************************************************     
IF seq.Step(50, TRUE, 'CAKNIE ODOSLANIE BLISTRU Z VYTAHU') THEN
    IF seq.IsFreshState THEN
        _timer(IN := FALSE);
    END_IF

	_outBufferIsWaitingEmpty:=TRUE;
	
    IF Components.PR14_Lift.AtHome AND_THEN
        Components.Q9_LiftConvRunReverse.IsTrue AND
        Components.Q6_OutgoingConvRun.Set() THEN
        _timer(in := Components.I14_PresentBlisterInLiftEnd.IsFalse AND Components.I15_PresentBlisterInLiftEntry.IsFalse,
            Pt := _config.StabilisationTime);

        IF _timer.Q THEN
            seq.CompleteStep();
        END_IF;
    END_IF;
END_IF

//***************************************************************************************************   

//***************************************************************************************************     
IF seq.Step(60, TRUE, 'CAKANIE BLISTA V POZICII  HORE PR5') THEN
    IF seq.IsFreshState THEN
        _timer(IN := FALSE);
    END_IF
	
    Components.Q6_OutgoingConvRun.Set();

    _timer(in := Components.I10_PresentBlisterAtOutgoingStopper1.Istrue, Pt := _config.StabilisationTime);
    IF _timer.Q THEN
        seq.CompleteStep();
    END_IF;

END_IF

//***************************************************************************************************   

//***************************************************************************************************     
IF seq.Step(70, TRUE, 'POLOZENIE BLISTROV NA NOVY BLISTER PR10 VYSUNUT PR11 ZASUNUT  A NASLEDNE PR7 ZASUNUT') THEN
    IF seq.IsFreshState THEN
        _timer(IN := FALSE);
    END_IF

    _timer(in := TRUE, Pt := T#5S);
    seq.StepCompleteWhen(Components.PR10_VerticalSepareOutgoingBlister1.MoveToWork().Done AND
            (Components.PR11_VerticalSepareOutgoingBlister2.MoveToHome().Done OR _timer.Q) AND_THEN
            Components.PR7_HorizontalSepareOutgoingBlisters.MoveToHome().Done);
END_IF

//***************************************************************************************************   

//***************************************************************************************************     
IF seq.Step(80, TRUE, 'KONTROLA POCTU VYSTUPNYCH BLISTROV') THEN
    messenger.Warning('ZASOBNIK NA VYSTUPNE BLISTRE PLNY!');
    Components.Q6_OutgoingConvRun.Set();

    IF Components.I12_OutgoingBufferIsFull.IsTrue AND Components.I13_OutgoingConveyorIsFull.IsFalse THEN
        seq.CompleteStep();
    ELSIF Components.I12_OutgoingBufferIsFull.IsFalse THEN
        seq.RequestStep(100);

    END_IF

END_IF

//***************************************************************************************************   

//***************************************************************************************************     
IF seq.Step(90, TRUE, 'ODOSLANIE PRAZDNYCH VYSTUPNYCH BLISTROV PR5 ZASUNUT') THEN
    IF seq.IsFreshState THEN
        _timer(IN := FALSE);
    END_IF

    _timer(In := Components.I10_PresentBlisterAtOutgoingStopper1.IsFalse, Pt := _config.StabilisationTime);

    IF Components.PR5_StopperConveyorOutgoing1.MoveToHome().Done AND_THEN
        Components.Q6_OutgoingConvRun.Set() AND_THEN
        _timer.Q then
        Seq.CompleteStep();
    END_IF;

END_IF

//***************************************************************************************************   

//***************************************************************************************************     
IF seq.Step(100, TRUE, 'VYSUNUTIE ZARAZKY PR5') THEN

    seq.StepCompleteWhen(Components.PR5_StopperConveyorOutgoing1.MoveToWork().Done);

END_IF

//***************************************************************************************************   

IF (seq.Step(inStepID := seq.RESTORE_STEP_ID,
    inEnabled := TRUE,
    inStepDescription := 'RETURN TO THE START OF THE SEQUENCE')) THEN
    //--------------------------------------------------------	
    refSequenceTask.DoneWhen(TRUE);
    seq.CompleteSequence();
    //--------------------------------------------------------			
END_IF;

IF refSequenceTask.HandleTaskError() THEN
    //here we can decide what to do
    _throwBlisterTask.Restore();

END_IF

seq.Close();
END_METHOD

METHOD PRIVATE SequenceResetToDefault
VAR_INPUT
	refSequenceTask : REFERENCE TO TcoFeedingSequenceTask;
	
	
END_VAR

VAR
    seq    : REFERENCE TO TcoCore.TcoSequence;

END_VAR

VAR_INST
	_timer:ton;
	
END_VAR
seq REF= refSequenceTask.Sequence;
refSequenceTask(inoStatus:=_status,inoConfig:=_config);
seq.Open();
seq.Observer := refSequenceTask.Observer;



		



//***************************************************************************************************     
//    This step will be executed and immediately finished, as the condition in Await method is true.
IF seq.Step(0,TRUE,'<#INIT#>') THEN   
	Messenger.Warning('<#BEZPECNOST ZARIADENIA NARUSENA. NIEJE MOZNE VYKONAT AKCIU#>');     
	IF _status.SafeCondition THEN
    	seq.CompleteStep();
	END_IF;
END_IF        
//***************************************************************************************************     



//***************************************************************************************************     
IF seq.Step(10,TRUE,'<#VYCHODIZA POLOHA - VYPNUTIE DOPRAVNIKOV#>') THEN   
	Components.Q4_EntryConvRun.Reset();
	Components.Q5_EntryConvRunReverse.Reset();
	Components.Q8_LiftConvRun.Reset();
	Components.Q9_LiftConvRunReverse.Reset();
	Components.Q6_OutgoingConvRun.Reset();
	Components.Q7_OutgoingConvRunReverse.Reset();
    seq.StepCompleteWhen(TRUE);
END_IF        
//***************************************************************************************************   


//***************************************************************************************************     
IF seq.Step(20,TRUE,'<#VYCHODIZA POLOHA - VYSUNUTIE ZARAZIEK PR1,PR3,PR4 A PR5#>') THEN   

    seq.StepCompleteWhen(Components.PR1_StopperConveyorEntry1.MoveToWork().Done 
		AND Components.PR3_StopperConveyorEntry3.MoveToWork().Done
		AND Components.PR4_StopperConveyorEntry4.MoveToWork().Done
		AND Components.PR5_StopperConveyorOutgoing1.MoveToWork().Done);
END_IF        
//***************************************************************************************************   

//***************************************************************************************************     
IF seq.Step(25,NOT _config.PR2_StopperConveyorEntry2Disabled,'<#VYCHODIZA POLOHA - VYSUNUTIE ZARAZKY PR2#>') THEN   

    seq.StepCompleteWhen(Components.PR2_StopperConveyorEntry2.MoveToWork().Done );
END_IF        
//***************************************************************************************************   
//***************************************************************************************************     
IF seq.Step(30,TRUE,'<#VYCHODIZA POLOHA - ZASUNUTIE PR6#>') THEN   


	    seq.StepCompleteWhen(Components.PR6_HorizontalSepareEntyBlisters.MoveToHome().Done);

END_IF        
//***************************************************************************************************   


//***************************************************************************************************     
IF seq.Step(40,TRUE,'<#VYCHODIZA POLOHA - VYSUNUTIE PR8#>') THEN   

	
	seq.StepCompleteWhen(Components.PR8_VerticalSepareEntryBlister1.MoveToHome().Done
		AND Components.PR9_VerticalSepareEntryBlister2.MoveToWork().Done);
		
END_IF        
//***************************************************************************************************  

//***************************************************************************************************     
IF seq.Step(50,NOT _config.PR12_HorizontalHoldEntryBlisterDisabled,'<#VYCHODIZA POLOHA - ZASUNUTIE PR12#>') THEN   

	
	seq.StepCompleteWhen(Components.PR12_HorizontalHoldEntryBlister.MoveToHome().Done);
		
END_IF        
//***************************************************************************************************   

//***************************************************************************************************     
IF seq.Step(55,TRUE,'<#VYCHODIZA POLOHA - ZASUNUTIE PR7#>') THEN   

	
	seq.StepCompleteWhen(Components.PR7_HorizontalSepareOutgoingBlisters.MoveToHome().Done);
		
END_IF        
//***************************************************************************************************   

//***************************************************************************************************     
IF seq.Step(60,TRUE,'<#VYCHODIZA POLOHA - VYSUNUTIE PR10 #>') THEN   

	
	seq.StepCompleteWhen(Components.PR10_VerticalSepareOutgoingBlister1.MoveToWork().Done);
		
END_IF        
//***************************************************************************************************   

//***************************************************************************************************     
IF seq.Step(70,TRUE,'<#VYCHODIZA POLOHA - VYSUNUTIE PR11 #>') THEN   

	
	seq.StepCompleteWhen(Components.PR11_VerticalSepareOutgoingBlister2.MoveToWork().Done);
		
END_IF        
//***************************************************************************************************   


//***************************************************************************************************     
IF seq.Step(80,TRUE,'<#VYCHODIZA POLOHA - VYSUNUTIE VYTAHU DO HORNEJ POZICIE PR14 #>') THEN   

	
	seq.StepCompleteWhen(Components.PR14_Lift.MoveToWork().Done);
		
END_IF        
//***************************************************************************************************   

//***************************************************************************************************     
IF seq.Step(90,TRUE,'<#VYCHODIZA POLOHA - CENTROVANIE KUSU VO VYHAHU VYSUNUTE PR13 #>') THEN   

	
	seq.StepCompleteWhen(Components.PR13_CenteringBlisterInLift.MoveToWork().Done);
		
END_IF        
//***************************************************************************************************  

IF (seq.Step(inStepID := seq.RESTORE_STEP_ID,
    inEnabled := TRUE,
    inStepDescription := 'RETURN TO THE START OF THE SEQUENCE')) THEN
    //--------------------------------------------------------	
		refSequenceTask.DoneWhen(TRUE);
    	seq.CompleteSequence();
    //--------------------------------------------------------			
END_IF;



IF refSequenceTask.HandleTaskError() THEN
	
	//here we can decide what to do
	//	refSequenceTask.Restore();

END_IF

seq.Close();
END_METHOD

(*~
	<docu>
		<summary>
		    Custom service (manual, maintenance) logic.
			This method must be implemented in derived class.
		</summary>			
	</docu>	
~*)
METHOD PROTECTED  ServiceMode
_components.Q3_AttentionSignalisationB.Service();
_components.Q2_AttentionSignalisationG.Service();
_components.Q1_AttentionSignalisationR.Service();
_components.PR13_CenteringBlisterInLift.Service();
_components.PR12_HorizontalHoldEntryBlister.Service();
_components.PR6_HorizontalSepareEntyBlisters.Service();
_components.PR14_Lift .Service();
_components.PR1_StopperConveyorEntry1 .Service();
_components.PR2_StopperConveyorEntry2.Service();
_components.PR3_StopperConveyorEntry3.Service();
_components.PR4_StopperConveyorEntry4.Service();
_components.PR5_StopperConveyorOutgoing1.Service();
_components.PR8_VerticalSepareEntryBlister1.Service();
_components.PR9_VerticalSepareEntryBlister2.Service();
_components.PR7_HorizontalSepareOutgoingBlisters.Service();
_components.PR10_VerticalSepareOutgoingBlister1.Service();
_components.PR11_VerticalSepareOutgoingBlister2.Service();
_components.Q4_EntryConvRun.Service();
_components.Q5_EntryConvRunReverse.Service();
_components.Q8_LiftConvRun.Service();
_components.Q9_LiftConvRunReverse.Service();
_components.Q6_OutgoingConvRun.Service();
_components.Q7_OutgoingConvRunReverse.Service();
END_METHOD

PROPERTY PUBLIC SetSequencesToStep : bool
GET
SetSequencesToStep:=_setSequencesToStep;
END_GET
SET
_setSequencesToStep:=SetSequencesToStep;
END_SET
END_PROPERTY

METHOD PUBLIC SetToDefault : TcoCore.ITcoTaskStatus
SetToDefault := _setToDefaultTask.Invoke();
END_METHOD

PROPERTY SetToDefaultTask : REFERENCE TO TcoFeedingSequenceTask
GET
SetToDefaultTask ref=_setToDefaultTask;
END_GET
END_PROPERTY

(*~
	<docu>
		<summary>
			Gets the status of the MTS Pls feeder. 					
		</summary>			
	</docu>	
~*)
PROPERTY Status : REFERENCE TO TcoPlrPaletizator_Status_v_1_x_x
GET
Status REF= _status;
END_GET
END_PROPERTY

METHOD PUBLIC ThrowBlister : TcoCore.ITcoTaskStatus
ThrowBlister := _throwBlisterTask.Invoke();
END_METHOD

PROPERTY ThrowBlisterTask : REFERENCE TO TcoFeedingSequenceTask
GET
ThrowBlisterTask ref=_throwBlisterTask;
END_GET
END_PROPERTY

END_FUNCTION_BLOCK

// ---- Abstractions/Components/MtsFeeding/Blisters/Pls/TcoPlsPaletizator.TcPOU
FUNCTION_BLOCK TcoPlsPaletizator EXTENDS TcoCore.TcoComponent
VAR_INPUT
    inSafeCondition : BOOL;
    inDoorOpen : BOOL;
END_VAR

VAR_OUTPUT
END_VAR
VAR
    {attribute addProperty Name "<#Config#>"}
    _config : TcoPlsPaletizator_Config_v_1_x_x;
    {attribute addProperty Name "<#Status#>"}
    {attribute clr [ReadOnly()]}
    _status : TcoPlsPaletizator_Status_v_1_x_x;
    {attribute addProperty Name "<#Control#>"}
    _control : TcoPlsPaletizator_Control_v_1_x_x;

    {attribute addProperty Name "<#Components#>"}
    _components : TcoPlsPaletizator_Components := (Parent := THIS^);

    {attribute addProperty Name "<#Poziadavka novy blister#>"}
    _feedNewBlisterTask : TcoFeedingSequenceTask(THIS^);
    {attribute addProperty Name "<#Poziadavka vylozenie blistera#>"}
    _throwBlisterTask : TcoFeedingSequenceTask(THIS^);
    {attribute addProperty Name "<#Poziadavka obsluhy vystupny buffer#>"}
    _hanldeOutBufferTask : TcoFeedingSequenceTask(THIS^);
    {attribute addProperty Name "<#Poziadavka vychodzej polohy#>"}
    _setToDefaultTask : TcoFeedingSequenceTask(THIS^);

    {attribute addProperty Name "<#Restore#>"}
    _restoreTask : TcoCore.TcoTask(THIS^);

    {attribute clr [CompilerOmits("BuilderPlainer", "BuilderOnliner","BuilderOnlinerInterface","BuilderShadowerInterface")]}
    _blinker : TcoBlinker(THIS^);
    _timerEntryEmpty : ton;
    _timerOutFull : ton;
    _timerDisableSafety : TON;
    {attribute addProperty Name "<#Temporarily disabled safety#>"}
    _temporarilyDisableSafety : BOOL;

    {attribute clr [CompilerOmits("BuilderPlainer", "BuilderOnliner","BuilderOnlinerInterface","BuilderShadowerInterface")]}
    restoreDone : BOOL;
    {attribute clr [CompilerOmits("BuilderPlainer", "BuilderOnliner","BuilderOnlinerInterface","BuilderShadowerInterface")]}
    _setSequencesToStep : BOOL := FALSE;
END_VAR

_status.SafeCondition := inSafeCondition;
Context.Environment.Messaging.Suspend();
_status.EntryBufferEmpty := NOT Components.I3_PresentBlistersInBufferEmpty.Signal;
_status.BlisterReady := Components.I4_PresentBlisterInWorkingPos.Signal AND Components.P7_SupportEntryBlister.AtWork;
_status.OutBufferFull := Components.I8_OutBlistersBufferIsFull.Signal;
Context.Environment.Messaging.Resume();

IF _config.StepModeManagableFromOutside THEN
    IF _setSequencesToStep THEN
        _feedNewBlisterTask.SetStepMode();
        _throwBlisterTask.SetStepMode();
        _hanldeOutBufferTask.SetStepMode();
        _setToDefaultTask.SetStepMode();
    ELSE
        _feedNewBlisterTask.SetCyclicMode();
        _throwBlisterTask.SetCyclicMode();
        _hanldeOutBufferTask.SetCyclicMode();
        _setToDefaultTask.SetCyclicMode();
    END_IF
END_IF;

_feedNewBlisterTask.Enabled := NOT _throwBlisterTask.Busy;
IF (_feedNewBlisterTask.Execute()) THEN
    SequenceIncomingBlister(refSequenceTask := _feedNewBlisterTask);
END_IF;

_throwBlisterTask.Enabled := NOT _feedNewBlisterTask.Busy;
IF (_throwBlisterTask.Execute()) THEN
    SequenceOutgoingBlister(refSequenceTask := _throwBlisterTask);
END_IF;

_hanldeOutBufferTask.Enabled := TRUE;
IF (_hanldeOutBufferTask.Execute()) THEN
    SequenceOutgoingBuffer(refSequenceTask := _hanldeOutBufferTask);
END_IF;

_setToDefaultTask.Enabled := TRUE;
IF (_setToDefaultTask.Execute()) THEN
    SequenceResetToDefault(refSequenceTask := _setToDefaultTask);
END_IF;

//*************RESTORE********************

_restoreTask.Enabled := TRUE;

IF _restoreTask.Execute() THEN
    Restore();
    _restoreTask.DoneWhen(inCondition := TRUE);
END_IF

//****************************************

//********************SAFETY******************
_timerDisableSafety(IN := _temporarilyDisableSafety, PT := _config.TimeToDisableSafety);

THIS^.Messenger.OnCondition(inCondition := _temporarilyDisableSafety).Warning('SAFTY TEMPORARILY DISABLED!');

IF NOT _temporarilyDisableSafety THEN

    Components.P7_SupportEntryBlister
        .SuspendMoveWorkExpression( Components.P7_SupportEntryBlister.MoveWorkTask.Busy AND NOT inSafeCondition, '<#Movement is blocked due safe zone is interupted(robot in zone)#>');

    Components.P7_SupportEntryBlister
        .SuspendMoveHomeExpression(Components.P7_SupportEntryBlister.MoveHomeTask.Busy AND NOT inSafeCondition, '<#Movement is blocked due safe zone is interupted(robot in zone)#>');

    Components.P8_FixEntryBlisterSide
        .SuspendMoveWorkExpression(Components.P8_FixEntryBlisterSide.MoveWorkTask.Busy AND NOT inSafeCondition, '<#Movement is blocked due safe zone is interupted(robot in zone)#>');

    Components.P8_FixEntryBlisterSide
        .SuspendMoveHomeExpression(Components.P8_FixEntryBlisterSide.MoveHomeTask.Busy AND NOT inSafeCondition, '<#Movement is blocked due safe zone is interupted(robot in zone)#>');

    IF NOT _config.LockBlisterInPickPosInactive THEN
        Components.P9_LockEntryBlisterTop
            .SuspendMoveWorkExpression(Components.P9_LockEntryBlisterTop.MoveWorkTask.Busy AND NOT inSafeCondition, '<#Movement is blocked due safe zone is interupted(robot in zone)#>');

        Components.P9_LockEntryBlisterTop
            .SuspendMoveHomeExpression(Components.P9_LockEntryBlisterTop.MoveHomeTask.Busy AND NOT inSafeCondition, '<#Movement is blocked due safe zone is interupted(robot in zone)#>');
    END_IF;

    Components.P4_FeedEntryBlister
        .SuspendMoveWorkExpression(NOT Components.P7_SupportEntryBlister.AtHome, 'Movement is blocked due P7 is not in home position');

    Components.P4_FeedEntryBlister
        .SuspendMoveHomeExpression(NOT Components.P6_VerticalSepareOutBlister.AtHome, 'Movement is blocked due P6 is not in home position');

    Components.P4_FeedEntryBlister
        .SuspendMoveHomeExpression(NOT Components.P5_HorizontalSepareOutBlisters.AtHome, 'Movement is blocked due P5 is not in home position');

    Components.P4_FeedEntryBlister
        .SuspendMoveHomeExpression(Components.I7_OutBlistersIsAboveOutBuffer.Signal, 'Movement is blocked due empty blister is not unloaded');

    Components.P7_SupportEntryBlister
        .SuspendMoveWorkExpression(NOT Components.P4_FeedEntryBlister.AtHome, 'Movement is blocked due P4 is not in home position');

    Components.P7_SupportEntryBlister
        .SuspendMoveWorkExpression(NOT Components.P4_FeedEntryBlister.AtHome, 'Movement is blocked due P4 is not in home position');
END_IF;

IF _timerDisableSafety.Q THEN
    _temporarilyDisableSafety := FALSE;
END_IF

PROPERTY Components : REFERENCE TO TcoPlsPaletizator_Components
GET
Components ref=_components;
END_GET
END_PROPERTY

(*~
	<docu>
		<summary>
			Gets the configuration of the MTS Pls feeder. 					
		</summary>			
	</docu>	
~*)
PROPERTY Config : REFERENCE TO TcoPlsPaletizator_Config_v_1_x_x
GET
Config REF= _config;
END_GET
END_PROPERTY

METHOD PUBLIC DefaultSignalisation
VAR_INPUT
END_VAR
Components.Q1_AttentionSignalisationR.Reset();
Components.Q2_AttentionSignalisationG.Reset();
Components.Q3_AttentionSignalisationB.Reset();

_blinker(inOffTime:=_config.BlinkTime,inOnTime:=_config.BlinkTime);
_timerEntryEmpty(in:= _status.EntryBufferEmpty,Pt:=_config.InfoTime);
_timerOutFull(in:=  _status.OutBufferFull ,Pt:=_config.InfoTime);
IF NOT inDoorOpen  
	AND NOT _timerEntryEmpty.Q
	AND NOT _timerOutFull.q THEN
	Components.Q2_AttentionSignalisationG.Set();
ELSIF  _blinker.IsOn THEN
	IF inDoorOpen AND 
		(
		THIS^._feedNewBlisterTask.Busy
		OR
		THIS^._throwBlisterTask.Busy
		OR
		THIS^._hanldeOutBufferTask.Busy )THEN
		Messenger.Warning('<#CAKANIE NA OBSLUHU PALETIZERA - ZAVRITE DVERE!#>');
		Components.Q1_AttentionSignalisationR.Set();
		Components.Q2_AttentionSignalisationG.Set();
	ELSIF _timerEntryEmpty.Q
		THEN
		Components.Q1_AttentionSignalisationR.Set();
		Components.Q2_AttentionSignalisationG.Set();
	ELSIF _timerOutFull.Q
		THEN
		
		Components.Q1_AttentionSignalisationR.Set();
		Components.Q2_AttentionSignalisationG.Set();

//	ELSIF NOT _status.OutBufferFull
//		AND _status.EntryBufferEmpty 
//		AND NOT _status.BlisterReady THEN	
//		Components.Q1_AttentionSignalisationR.Set();
//	ELSIF  _status.OutBufferFull  THEN
//		Components.Q1_AttentionSignalisationR.Set();	
	
	END_IF;


	
END_IF;
END_METHOD

METHOD PUBLIC FeedNewBlister : TcoCore.ITcoTaskStatus

FeedNewBlister := _feedNewBlisterTask.Invoke();
END_METHOD

PROPERTY FeedNewBlisterTask : REFERENCE TO TcoFeedingSequenceTask
GET
FeedNewBlisterTask ref=_feedNewBlisterTask;
END_GET
END_PROPERTY

PROPERTY HandleOutBufferTask : REFERENCE TO TcoFeedingSequenceTask
GET
HandleOutBufferTask ref=_hanldeOutBufferTask;
END_GET
END_PROPERTY

PROPERTY OutBufferFull : bool
GET
OutBufferFull:=_status.OutBufferFull;
END_GET
END_PROPERTY

PROPERTY ReadyToUnloadComponent : bool
GET
ReadyToUnloadComponent:=_status.BlisterReady;
END_GET
END_PROPERTY

(*~
	<docu>
		<summary>
			Restores this instance to the Ready state. Can be called explicitly or from within one of the restore mechanisms.	
		</summary>			
	</docu>	
~*)
METHOD  Restore : ITcoRestorable
_hanldeOutBufferTask.Restore();
_feedNewBlisterTask.Restore();
_throwBlisterTask.Restore();
_setToDefaultTask.Restore();
_messenger.UnPin();
END_METHOD

METHOD PRIVATE SequenceIncomingBlister
VAR_INPUT
	refSequenceTask : REFERENCE TO TcoFeedingSequenceTask;
	
	
END_VAR

VAR
    seq    : REFERENCE TO TcoCore.TcoSequence;


END_VAR
seq REF= refSequenceTask.Sequence;
refSequenceTask(inoStatus:=_status,inoConfig:=_config);


seq.Open();
seq.Observer := refSequenceTask.Observer;



		



//***************************************************************************************************     
//    This step will be executed and immediately finished, as the condition in Await method is true.
IF seq.Step(0,TRUE,'<#INIT#>') THEN   
	Messenger.Warning('<#BEZPECNOST ZARIADENIA NARUSENA. NIEJE MOZNE VYKONAT AKCIU#>');     
	IF _status.SafeCondition THEN
    	seq.CompleteStep();
	END_IF;
END_IF        
//***************************************************************************************************     

 
//***************************************************************************************************     
IF seq.Step(10,TRUE,'<#KONTROLA POCTU VSTUPNYCH BLISTROV#>') THEN   
    Messenger.Warning('<#PODAVAC PRAZDNY! DOPLNE VSTUPNE BLISTRE !#>');
    seq.StepCompleteWhen(Components.I3_PresentBlistersInBufferEmpty.IsTrue);
END_IF        
//***************************************************************************************************     


        
//***************************************************************************************************     
IF seq.Step(20,TRUE,'<#SEPAROVANIE VSTUPNEHO BLISTRA - VERTIKALNE VALCE VYSUNUTE P1 A P2 #>') THEN   

    seq.StepCompleteWhen(THIS^.Components.P1_VerticalSepareEntryBlisters.MoveToWork().Done AND THIS^.Components.P2_VerticalSepareEntryBlisters.MoveToWork().Done);
END_IF        
//***************************************************************************************************     


//***************************************************************************************************     
IF seq.Step(30,TRUE,'<#SEPAROVANIE VSTUPNEHO BLISTRA - SEPAROVANIE ZASUNUTE P3#>') THEN   

    seq.StepCompleteWhen(THIS^.Components.P3_HorizontalSepareEntryBlisters.MoveToHome().Done);
END_IF        
//***************************************************************************************************     


//***************************************************************************************************     
IF seq.Step(40,TRUE,'<#SEPAROVANIE VSTUPNEHO BLISTRA - VERTIKALNE VALCE  ZASUNUT P1#>') THEN   

    seq.StepCompleteWhen(THIS^.Components.P1_VerticalSepareEntryBlisters.MoveToHome().Done );
END_IF        
//***************************************************************************************************     

//***************************************************************************************************     
IF seq.Step(45,TRUE,'<#SEPAROVANIE VSTUPNEHO BLISTRA - VERTIKALNE VALCE VYSUNUT P2#>') THEN   

    seq.StepCompleteWhen( THIS^.Components.P2_VerticalSepareEntryBlisters.MoveToWork().Done);
END_IF        
//***************************************************************************************************     


//***************************************************************************************************     
IF seq.Step(50,TRUE,'<#SEPAROVANIE VSTUPNEHO BLISTRA - SEPAROVANIE VYSUNUTE P3 A P10#>') THEN   

    seq.StepCompleteWhen(THIS^.Components.P3_HorizontalSepareEntryBlisters.MoveToWork().Done AND (Components.P10_HoldEntrySepareOutBlister.MoveToWork().Done or _config.SepareBlistersAtEntryInactive));
END_IF        
//***************************************************************************************************     

//***************************************************************************************************     
IF seq.Step(60,TRUE,'<#SEPAROVANIE VSTUPNEHO BLISTRA - VERTIKALNE VALCE ZASUNUT P1 A P@#>') THEN   

    seq.StepCompleteWhen(THIS^.Components.P1_VerticalSepareEntryBlisters.MoveToHome().Done AND THIS^.Components.P2_VerticalSepareEntryBlisters.MoveToHome().Done); 
					
END_IF        
//***************************************************************************************************     

//***************************************************************************************************     
IF seq.Step(65,NOT _config.SepareBlistersAtEntryInactive,'<#SEPAROVANIE VSTUPNEHO BLISTRA - ZASUNUTIE P10>') THEN   

    seq.StepCompleteWhen(Components.P10_HoldEntrySepareOutBlister.MoveToHome().Done  );
END_IF        
//***************************************************************************************************     

//***************************************************************************************************   
IF seq.Step(70,TRUE,'<#KONTROLA PRITOMNOSTI SEPAROVANEHO KUSU#>') THEN   
    Messenger.Error('<#PODAVAC PRAZDNY! DOPLNE BLISTRE !#>');
    seq.StepCompleteWhen(THIS^.Components.I1_PresentBlisterEntry.IsTrue AND (THIS^.Components.I2_PresentBlisterEntryEmptySpace.IsTrue) );
END_IF        
//***************************************************************************************************     


//***************************************************************************************************     
IF seq.Step(80,TRUE,'<#SEPAROVANIE VSTUPNEHO BLISTRA - UPEVNENIE BLISTRA ZASUNUT P8#>') THEN   

    seq.StepCompleteWhen(THIS^.Components.P8_FixEntryBlisterSide.MoveToHome().Done);
END_IF        
//***************************************************************************************************     

//***************************************************************************************************     
IF seq.Step(85,TRUE,'<#SEPAROVANIE VSTUPNEHO BLISTRA - CAKANIE NA PRESUNUTIE BLISTRA DO ODOBERACEJ POLOHY P4 A I1 #>') THEN   

    seq.StepCompleteWhen(THIS^.Components.P4_FeedEntryBlister.MoveToWork().Done AND Components.i4_PresentBlisterInWorkingPos.IsTrue);
END_IF        
//***************************************************************************************************     


//***************************************************************************************************     
IF seq.Step(90,TRUE,'<#SEPAROVANIE VSTUPNEHO BLISTRA - UPEVENIE BLISTRA ZBOKU#>') THEN   

    seq.StepCompleteWhen(THIS^.Components.P8_FixEntryBlisterSide.MoveToWork().Done);
END_IF        
//***************************************************************************************************     



//***************************************************************************************************     
IF seq.Step(100,TRUE,'<#SEPAROVANIE VSTUPNEHO BLISTRA - NPRESUNUTIE BLISTRA DO POZICIE NABERANIA#>') THEN   

   IF THIS^.Components.P6_VerticalSepareOutBlister.AtHome THEN
	    seq.CompleteStep();
	ELSE
		Messenger.Error('VYSTUPNY BUFFER NIEJE V HORNEJ POZICII!(P6)');
	END_IF
END_IF        
//***************************************************************************************************   

//***************************************************************************************************     
IF seq.Step(110,TRUE,'<#SEPAROVANIE VSTUPNEHO BLISTRA - ZASUNUTE P4#>') THEN   

	 seq.StepCompleteWhen(THIS^.Components.P4_FeedEntryBlister.MoveToHome().Done) ;
	
END_IF        
//***************************************************************************************************   


//***************************************************************************************************     
IF seq.Step(120,TRUE,'<#SEPAROVANIE VSTUPNEHO BLISTRA - PODoPRETIE  A ZAFIXOVANIE KUSU P7 VYSUNT A P9 ZASUNUT #>') THEN   

    seq.StepCompleteWhen(THIS^.Components.P7_SupportEntryBlister.MoveToWork().Done AND (THIS^.Components.P9_LockEntryBlisterTop.MoveToHome().Done OR _config.LockBlisterInPickPosInactive));
END_IF        
//***************************************************************************************************   




